LIN {X 0,Y 459.073,Z 809.06,A -85,B 0,C 180,E1 14501.398,E2 14501.398} C_VEL
LIN {X 0,Y 458.818,Z 809.06,A -85,B 0,C 180,E1 14507.25,E2 14507.25} C_VEL
LIN {X 0,Y 458.467,Z 809.06,A -85,B 0,C 180,E1 14513.306,E2 14513.306} C_VEL
LIN {X 0,Y 458.275,Z 809.06,A -85,B 0,C 180,E1 14519.651,E2 14519.651} C_VEL
LIN {X 0,Y 458.077,Z 809.06,A -85,B 0,C 180,E1 14526.434,E2 14526.434} C_VEL
LIN {X 0,Y 458.07,Z 809.06,A -85,B 0,C 180,E1 14531.291,E2 14531.291} C_VEL
LIN {X 0,Y 458.072,Z 809.06,A -85,B 0,C 180,E1 14536.54,E2 14536.54} C_VEL
LIN {X 0,Y 458,Z 809.06,A -85,B 0,C 180,E1 14542.368,E2 14542.368} C_VEL
LIN {X 0,Y 458.221,Z 809.06,A -85,B 0,C 180,E1 14549.039,E2 14549.039} C_VEL
LIN {X 0,Y 458.429,Z 809.06,A -85,B 0,C 180,E1 14554.63,E2 14554.63} C_VEL
LIN {X 0,Y 458.704,Z 809.06,A -85,B 0,C 180,E1 14560.768,E2 14560.768} C_VEL
LIN {X 0,Y 458.946,Z 809.06,A -85,B 0,C 180,E1 14566.677,E2 14566.677} C_VEL
LIN {X 0,Y 459.248,Z 809.06,A -85,B 0,C 180,E1 14573.134,E2 14573.134} C_VEL
LIN {X 0,Y 459.567,Z 809.06,A -85,B 0,C 180,E1 14578.117,E2 14578.117} C_VEL
LIN {X 0,Y 459.486,Z 809.06,A -85,B 0,C 180,E1 14583.772,E2 14583.772} C_VEL
LIN {X 0,Y 459.188,Z 809.06,A -85,B 0,C 180,E1 14589.471,E2 14589.471} C_VEL
LIN {X 0,Y 458.841,Z 809.06,A -85,B 0,C 180,E1 14595.275,E2 14595.275} C_VEL
LIN {X 0,Y 458.62,Z 809.313,A -85,B 0,C 180,E1 14601.041,E2 14601.041} C_VEL
LIN {X 0,Y 460.727,Z 814.529,A -85,B 0,C 180,E1 14601.677,E2 14601.677} C_VEL
LIN {X 0,Y 463.517,Z 818.136,A -85,B 0,C 180,E1 14602.358,E2 14602.358} C_VEL
LIN {X 0,Y 484.639,Z 848.609,A -85,B 0,C 180,E1 14607.191,E2 14607.191} C_VEL
LIN {X 0,Y 509.827,Z 888.021,A -85,B 0,C 180,E1 14612.178,E2 14612.178} C_VEL
LIN {X 0,Y 531.176,Z 928.04,A -85,B 0,C 180,E1 14616.332,E2 14616.332} C_VEL
LIN {X 0,Y 533.852,Z 935.082,A -85,B 0,C 180,E1 14616.915,E2 14616.915} C_VEL
LIN {X 0,Y 525.994,Z 983.884,A -85,B 0,C 180,E1 14618.511,E2 14618.511} C_VEL
LIN {X 0,Y 516.792,Z 1031.445,A -85,B 0,C 180,E1 14620.799,E2 14620.799} C_VEL
LIN {X 0,Y 506.374,Z 1076.578,A -85,B 0,C 180,E1 14623.742,E2 14623.742} C_VEL
LIN {X 0,Y 495.446,Z 1119.708,A -85,B 0,C 180,E1 14627.415,E2 14627.415} C_VEL
LIN {X 0,Y 484.874,Z 1160.046,A -85,B 0,C 180,E1 14631.936,E2 14631.936} C_VEL
LIN {X 0,Y 476.093,Z 1194.068,A -85,B 0,C 180,E1 14636.796,E2 14636.796} C_VEL
LIN {X 0,Y 468.636,Z 1225.613,A -85,B 0,C 180,E1 14642.62,E2 14642.62} C_VEL
LIN {X 0,Y 464.052,Z 1248.469,A -85,B 0,C 180,E1 14648.117,E2 14648.117} C_VEL
LIN {X 0,Y 461.344,Z 1266.286,A -85,B 0,C 180,E1 14653.827,E2 14653.827} C_VEL
LIN {X 0,Y 459.993,Z 1278.774,A -85,B 0,C 180,E1 14659.554,E2 14659.554} C_VEL
LIN {X 0,Y 459.672,Z 1284.621,A -85,B 0,C 180,E1 14664.333,E2 14664.333} C_VEL
LIN {X 0,Y 459.56,Z 1286.34,A -85,B 0,C 180,E1 14667.341,E2 14667.341} C_VEL
LIN {X 0,Y 457.078,Z 1286.869,A -85,B 0,C 180,E1 14668.953,E2 14668.953} C_VEL
LIN {X 0,Y 451.946,Z 1286.314,A -85,B 0,C 180,E1 14671.378,E2 14671.378} C_VEL
LIN {X 0,Y 451.892,Z 1286.241,A -85,B 0,C 180,E1 14671.658,E2 14671.658} C_VEL
LIN {X 0,Y 451.956,Z 1281.773,A -85,B 0,C 180,E1 14677.677,E2 14677.677} C_VEL
LIN {X 0,Y 452.703,Z 1272.747,A -85,B 0,C 180,E1 14683.013,E2 14683.013} C_VEL
LIN {X 0,Y 454.412,Z 1258.506,A -85,B 0,C 180,E1 14688.449,E2 14688.449} C_VEL
LIN {X 0,Y 457.628,Z 1239.088,A -85,B 0,C 180,E1 14693.825,E2 14693.825} C_VEL
LIN {X 0,Y 462.745,Z 1212.947,A -85,B 0,C 180,E1 14699.319,E2 14699.319} C_VEL
LIN {X 0,Y 469.367,Z 1182.336,A -85,B 0,C 180,E1 14704.276,E2 14704.276} C_VEL
LIN {X 0,Y 477.757,Z 1144.374,A -85,B 0,C 180,E1 14709.083,E2 14709.083} C_VEL
LIN {X 0,Y 486.62,Z 1104.059,A -85,B 0,C 180,E1 14713.08,E2 14713.08} C_VEL
LIN {X 0,Y 496.53,Z 1056.093,A -85,B 0,C 180,E1 14716.748,E2 14716.748} C_VEL
LIN {X 0,Y 505.91,Z 1006.434,A -85,B 0,C 180,E1 14719.639,E2 14719.639} C_VEL
LIN {X 0,Y 515.783,Z 948.619,A -85,B 0,C 180,E1 14722.104,E2 14722.104} C_VEL
LIN {X 0,Y 517.829,Z 935.284,A -85,B 0,C 180,E1 14722.543,E2 14722.543} C_VEL
LIN {X 0,Y 507.618,Z 899.519,A -85,B 0,C 180,E1 14726.042,E2 14726.042} C_VEL
LIN {X 0,Y 505.964,Z 885.962,A -85,B 0,C 180,E1 14728.048,E2 14728.048} C_VEL
LIN {X 0,Y 505.994,Z 884.666,A -85,B 0,C 180,E1 14728.412,E2 14728.412} C_VEL
LIN {X 0,Y 504.35,Z 894.37,A -85,B 0,C 180,E1 14730.603,E2 14730.603} C_VEL
LIN {X 0,Y 507.893,Z 921.665,A -85,B 0,C 180,E1 14734.702,E2 14734.702} C_VEL
LIN {X 0,Y 511.089,Z 938.057,A -85,B 0,C 180,E1 14736.979,E2 14736.979} C_VEL
LIN {X 0,Y 500.885,Z 977.012,A -85,B 0,C 180,E1 14740.046,E2 14740.046} C_VEL
LIN {X 0,Y 489.61,Z 1013.591,A -85,B 0,C 180,E1 14743.873,E2 14743.873} C_VEL
LIN {X 0,Y 479.089,Z 1044.899,A -85,B 0,C 180,E1 14748.178,E2 14748.178} C_VEL
LIN {X 0,Y 468.845,Z 1074.319,A -85,B 0,C 180,E1 14753.523,E2 14753.523} C_VEL
LIN {X 0,Y 460.77,Z 1098.348,A -85,B 0,C 180,E1 14759.515,E2 14759.515} C_VEL
LIN {X 0,Y 455.737,Z 1115.395,A -85,B 0,C 180,E1 14765.369,E2 14765.369} C_VEL
LIN {X 0,Y 453.06,Z 1127.764,A -85,B 0,C 180,E1 14771.542,E2 14771.542} C_VEL
LIN {X 0,Y 451.778,Z 1135.121,A -85,B 0,C 180,E1 14777.517,E2 14777.517} C_VEL
LIN {X 0,Y 450.908,Z 1138.251,A -85,B 0,C 180,E1 14783.71,E2 14783.71} C_VEL
LIN {X 0,Y 451.301,Z 1136.637,A -85,B 0,C 180,E1 14790.146,E2 14790.146} C_VEL
LIN {X 0,Y 452.358,Z 1131.437,A -85,B 0,C 180,E1 14795.485,E2 14795.485} C_VEL
LIN {X 0,Y 453.774,Z 1122.657,A -85,B 0,C 180,E1 14800.796,E2 14800.796} C_VEL
LIN {X 0,Y 456.953,Z 1108.165,A -85,B 0,C 180,E1 14806.673,E2 14806.673} C_VEL
LIN {X 0,Y 462.638,Z 1088.104,A -85,B 0,C 180,E1 14812.52,E2 14812.52} C_VEL
LIN {X 0,Y 470.74,Z 1062.034,A -85,B 0,C 180,E1 14818.105,E2 14818.105} C_VEL
LIN {X 0,Y 480.037,Z 1033.327,A -85,B 0,C 180,E1 14822.802,E2 14822.802} C_VEL
LIN {X 0,Y 491.09,Z 998.255,A -85,B 0,C 180,E1 14827.17,E2 14827.17} C_VEL
LIN {X 0,Y 502.007,Z 960.535,A -85,B 0,C 180,E1 14830.786,E2 14830.786} C_VEL
LIN {X 0,Y 508.357,Z 935.557,A -85,B 0,C 180,E1 14832.715,E2 14832.715} C_VEL
LIN {X 0,Y 498.985,Z 904.371,A -85,B 0,C 180,E1 14836.88,E2 14836.88} C_VEL
LIN {X 0,Y 485.509,Z 871.059,A -85,B 0,C 180,E1 14841.568,E2 14841.568} C_VEL
LIN {X 0,Y 469.62,Z 840.002,A -85,B 0,C 180,E1 14846.422,E2 14846.422} C_VEL
LIN {X 0,Y 454.416,Z 815.01,A -85,B 0,C 180,E1 14850.902,E2 14850.902} C_VEL
LIN {X 0,Y 451.695,Z 809.882,A -85,B 0,C 180,E1 14851.745,E2 14851.745} C_VEL
LIN {X 0,Y 451.507,Z 809.06,A -85,B 0,C 180,E1 14853.846,E2 14853.846} C_VEL
LIN {X 0,Y 451.253,Z 809.06,A -85,B 0,C 180,E1 14859.646,E2 14859.646} C_VEL
LIN {X 0,Y 450.953,Z 809.06,A -85,B 0,C 180,E1 14865.557,E2 14865.557} C_VEL
LIN {X 0,Y 450.624,Z 809.06,A -85,B 0,C 180,E1 14871.653,E2 14871.653} C_VEL
LIN {X 0,Y 450.391,Z 809.06,A -85,B 0,C 180,E1 14878.023,E2 14878.023} C_VEL
LIN {X 0,Y 450.197,Z 809.06,A -85,B 0,C 180,E1 14884.801,E2 14884.801} C_VEL
LIN {X 0,Y 450.133,Z 809.06,A -85,B 0,C 180,E1 14889.639,E2 14889.639} C_VEL
LIN {X 0,Y 450.084,Z 809.06,A -85,B 0,C 180,E1 14895.172,E2 14895.172} C_VEL
LIN {X 0,Y 450.079,Z 809.06,A -85,B 0,C 180,E1 14900.562,E2 14900.562} C_VEL
LIN {X 0,Y 450.156,Z 809.06,A -85,B 0,C 180,E1 14907.068,E2 14907.068} C_VEL
LIN {X 0,Y 450.393,Z 809.06,A -85,B 0,C 180,E1 14911.988,E2 14911.988} C_VEL
LIN {X 0,Y 450.672,Z 809.06,A -85,B 0,C 180,E1 14918.359,E2 14918.359} C_VEL
LIN {X 0,Y 450.885,Z 809.06,A -85,B 0,C 180,E1 14924.45,E2 14924.45} C_VEL
LIN {X 0,Y 451.262,Z 809.06,A -85,B 0,C 180,E1 14930.363,E2 14930.363} C_VEL
LIN {X 0,Y 451.566,Z 809.06,A -85,B 0,C 180,E1 14936.164,E2 14936.164} C_VEL
LIN {X 0,Y 451.767,Z 809.06,A -85,B 0,C 180,E1 14941.917,E2 14941.917} C_VEL
LIN {X 0,Y 451.343,Z 809.06,A -85,B 0,C 180,E1 14947.696,E2 14947.696} C_VEL
LIN {X 0,Y 451.023,Z 809.06,A -85,B 0,C 180,E1 14953.661,E2 14953.661} C_VEL
LIN {X 0,Y 450.817,Z 809.82,A -85,B 0,C 180,E1 14959.392,E2 14959.392} C_VEL
LIN {X 0,Y 453.497,Z 815.064,A -85,B 0,C 180,E1 14960.162,E2 14960.162} C_VEL
LIN {X 0,Y 455.851,Z 818.218,A -85,B 0,C 180,E1 14960.792,E2 14960.792} C_VEL
LIN {X 0,Y 474.523,Z 845.268,A -85,B 0,C 180,E1 14965.35,E2 14965.35} C_VEL
LIN {X 0,Y 499.268,Z 883.021,A -85,B 0,C 180,E1 14970.523,E2 14970.523} C_VEL
LIN {X 0,Y 521.728,Z 923.677,A -85,B 0,C 180,E1 14975.016,E2 14975.016} C_VEL
LIN {X 0,Y 528.094,Z 937.427,A -85,B 0,C 180,E1 14976.349,E2 14976.349} C_VEL
LIN {X 0,Y 519.566,Z 988.021,A -85,B 0,C 180,E1 14978.079,E2 14978.079} C_VEL
LIN {X 0,Y 510.247,Z 1034.148,A -85,B 0,C 180,E1 14980.364,E2 14980.364} C_VEL
LIN {X 0,Y 498.846,Z 1081.49,A -85,B 0,C 180,E1 14983.565,E2 14983.565} C_VEL
LIN {X 0,Y 487.789,Z 1123.072,A -85,B 0,C 180,E1 14987.26,E2 14987.26} C_VEL
LIN {X 0,Y 477.179,Z 1162.261,A -85,B 0,C 180,E1 14991.785,E2 14991.785} C_VEL
LIN {X 0,Y 468.218,Z 1195.558,A -85,B 0,C 180,E1 14996.718,E2 14996.718} C_VEL
LIN {X 0,Y 461.085,Z 1224.685,A -85,B 0,C 180,E1 15002.228,E2 15002.228} C_VEL
LIN {X 0,Y 456.204,Z 1248.219,A -85,B 0,C 180,E1 15008.033,E2 15008.033} C_VEL
LIN {X 0,Y 453.562,Z 1265.022,A -85,B 0,C 180,E1 15013.542,E2 15013.542} C_VEL
LIN {X 0,Y 452.345,Z 1275.819,A -85,B 0,C 180,E1 15018.43,E2 15018.43} C_VEL
LIN {X 0,Y 451.967,Z 1281.836,A -85,B 0,C 180,E1 15022.307,E2 15022.307} C_VEL
LIN {X 0,Y 451.745,Z 1286.16,A -85,B 0,C 180,E1 15028.075,E2 15028.075} C_VEL
LIN {X 0,Y 451.892,Z 1286.241,A -85,B 0,C 180,E1 15031.658,E2 15031.658} C_VEL
LIN {X 0,Y 449.493,Z 1285.263,A -85,B 0,C 180,E1 15033.286,E2 15033.286} C_VEL
LIN {X 0,Y 444.015,Z 1282.245,A -85,B 0,C 180,E1 15036.001,E2 15036.001} C_VEL
LIN {X 0,Y 444.472,Z 1275.955,A -85,B 0,C 180,E1 15040.768,E2 15040.768} C_VEL
LIN {X 0,Y 445.669,Z 1264.065,A -85,B 0,C 180,E1 15046.235,E2 15046.235} C_VEL
LIN {X 0,Y 448.266,Z 1246.87,A -85,B 0,C 180,E1 15051.756,E2 15051.756} C_VEL
LIN {X 0,Y 452.324,Z 1224.795,A -85,B 0,C 180,E1 15057.066,E2 15057.066} C_VEL
LIN {X 0,Y 458.574,Z 1196.263,A -85,B 0,C 180,E1 15062.373,E2 15062.373} C_VEL
LIN {X 0,Y 466.395,Z 1162.049,A -85,B 0,C 180,E1 15067.294,E2 15067.294} C_VEL
LIN {X 0,Y 475.604,Z 1121.839,A -85,B 0,C 180,E1 15071.841,E2 15071.841} C_VEL
LIN {X 0,Y 485.521,Z 1077.379,A -85,B 0,C 180,E1 15075.699,E2 15075.699} C_VEL
LIN {X 0,Y 495.288,Z 1029.918,A -85,B 0,C 180,E1 15078.903,E2 15078.903} C_VEL
LIN {X 0,Y 504.786,Z 979.028,A -85,B 0,C 180,E1 15081.496,E2 15081.496} C_VEL
LIN {X 0,Y 511.598,Z 937.834,A -85,B 0,C 180,E1 15083.138,E2 15083.138} C_VEL
LIN {X 0,Y 503.854,Z 906.093,A -85,B 0,C 180,E1 15086.378,E2 15086.378} C_VEL
LIN {X 0,Y 503.15,Z 893.729,A -85,B 0,C 180,E1 15088.205,E2 15088.205} C_VEL
LIN {X 0,Y 503.056,Z 893.125,A -85,B 0,C 180,E1 15088.555,E2 15088.555} C_VEL
LIN {X 0,Y 500.921,Z 904.138,A -85,B 0,C 180,E1 15090.847,E2 15090.847} C_VEL
LIN {X 0,Y 505.503,Z 941.412,A -85,B 0,C 180,E1 15096.443,E2 15096.443} C_VEL
LIN {X 0,Y 494.875,Z 980.106,A -85,B 0,C 180,E1 15099.56,E2 15099.56} C_VEL
LIN {X 0,Y 483.27,Z 1016.326,A -85,B 0,C 180,E1 15103.422,E2 15103.422} C_VEL
LIN {X 0,Y 472.262,Z 1047.658,A -85,B 0,C 180,E1 15107.819,E2 15107.819} C_VEL
LIN {X 0,Y 462.173,Z 1075.434,A -85,B 0,C 180,E1 15112.957,E2 15112.957} C_VEL
LIN {X 0,Y 454.375,Z 1097.488,A -85,B 0,C 180,E1 15118.443,E2 15118.443} C_VEL
LIN {X 0,Y 448.592,Z 1115.922,A -85,B 0,C 180,E1 15124.658,E2 15124.658} C_VEL
LIN {X 0,Y 445.664,Z 1127.858,A -85,B 0,C 180,E1 15130.543,E2 15130.543} C_VEL
LIN {X 0,Y 444.326,Z 1134.908,A -85,B 0,C 180,E1 15135.786,E2 15135.786} C_VEL
LIN {X 0,Y 443.237,Z 1139.205,A -85,B 0,C 180,E1 15142.023,E2 15142.023} C_VEL
LIN {X 0,Y 443.275,Z 1138.821,A -85,B 0,C 180,E1 15148.503,E2 15148.503} C_VEL
LIN {X 0,Y 444.258,Z 1134.571,A -85,B 0,C 180,E1 15153.963,E2 15153.963} C_VEL
LIN {X 0,Y 445.795,Z 1125.624,A -85,B 0,C 180,E1 15160.089,E2 15160.089} C_VEL
LIN {X 0,Y 448.665,Z 1112.355,A -85,B 0,C 180,E1 15165.931,E2 15165.931} C_VEL
LIN {X 0,Y 454.479,Z 1092.107,A -85,B 0,C 180,E1 15172.18,E2 15172.18} C_VEL
LIN {X 0,Y 461.863,Z 1069.016,A -85,B 0,C 180,E1 15177.464,E2 15177.464} C_VEL
LIN {X 0,Y 472.192,Z 1038.17,A -85,B 0,C 180,E1 15182.773,E2 15182.773} C_VEL
LIN {X 0,Y 482.736,Z 1006.027,A -85,B 0,C 180,E1 15186.992,E2 15186.992} C_VEL
LIN {X 0,Y 494.625,Z 966.727,A -85,B 0,C 180,E1 15190.932,E2 15190.932} C_VEL
LIN {X 0,Y 502.079,Z 938.758,A -85,B 0,C 180,E1 15193.169,E2 15193.169} C_VEL
LIN {X 0,Y 492.985,Z 907.827,A -85,B 0,C 180,E1 15197.393,E2 15197.393} C_VEL
LIN {X 0,Y 480.041,Z 875.321,A -85,B 0,C 180,E1 15202.092,E2 15202.092} C_VEL
LIN {X 0,Y 464.938,Z 845.25,A -85,B 0,C 180,E1 15206.922,E2 15206.922} C_VEL
LIN {X 0,Y 450.629,Z 821.483,A -85,B 0,C 180,E1 15211.276,E2 15211.276} C_VEL
LIN {X 0,Y 446.35,Z 814.995,A -85,B 0,C 180,E1 15212.615,E2 15212.615} C_VEL
LIN {X 0,Y 443.672,Z 810.022,A -85,B 0,C 180,E1 15213.486,E2 15213.486} C_VEL
LIN {X 0,Y 443.596,Z 809.06,A -85,B 0,C 180,E1 15213.914,E2 15213.914} C_VEL
LIN {X 0,Y 443.332,Z 809.06,A -85,B 0,C 180,E1 15219.82,E2 15219.82} C_VEL
LIN {X 0,Y 443.006,Z 809.06,A -85,B 0,C 180,E1 15225.843,E2 15225.843} C_VEL
LIN {X 0,Y 442.652,Z 809.06,A -85,B 0,C 180,E1 15232.064,E2 15232.064} C_VEL
LIN {X 0,Y 442.457,Z 809.06,A -85,B 0,C 180,E1 15238.572,E2 15238.572} C_VEL
LIN {X 0,Y 442.267,Z 809.06,A -85,B 0,C 180,E1 15245.518,E2 15245.518} C_VEL
LIN {X 0,Y 442.109,Z 809.06,A -85,B 0,C 180,E1 15251.247,E2 15251.247} C_VEL
LIN {X 0,Y 442.089,Z 809.06,A -85,B 0,C 180,E1 15256.878,E2 15256.878} C_VEL
LIN {X 0,Y 442.109,Z 809.06,A -85,B 0,C 180,E1 15262.036,E2 15262.036} C_VEL
LIN {X 0,Y 442.287,Z 809.06,A -85,B 0,C 180,E1 15268.677,E2 15268.677} C_VEL
LIN {X 0,Y 442.506,Z 809.06,A -85,B 0,C 180,E1 15273.648,E2 15273.648} C_VEL
LIN {X 0,Y 442.832,Z 809.06,A -85,B 0,C 180,E1 15280.05,E2 15280.05} C_VEL
LIN {X 0,Y 443.096,Z 809.06,A -85,B 0,C 180,E1 15286.191,E2 15286.191} C_VEL
LIN {X 0,Y 443.431,Z 809.06,A -85,B 0,C 180,E1 15292.167,E2 15292.167} C_VEL
LIN {X 0,Y 443.778,Z 809.06,A -85,B 0,C 180,E1 15298.05,E2 15298.05} C_VEL
LIN {X 0,Y 443.661,Z 809.06,A -85,B 0,C 180,E1 15303.906,E2 15303.906} C_VEL
LIN {X 0,Y 443.324,Z 809.06,A -85,B 0,C 180,E1 15309.813,E2 15309.813} C_VEL
LIN {X 0,Y 442.959,Z 809.06,A -85,B 0,C 180,E1 15315.837,E2 15315.837} C_VEL
LIN {X 0,Y 442.983,Z 809.793,A -85,B 0,C 180,E1 15317.595,E2 15317.595} C_VEL
LIN {X 0,Y 445.55,Z 814.971,A -85,B 0,C 180,E1 15318.432,E2 15318.432} C_VEL
LIN {X 0,Y 447.849,Z 817.771,A -85,B 0,C 180,E1 15319.064,E2 15319.064} C_VEL
LIN {X 0,Y 470.21,Z 850.079,A -85,B 0,C 180,E1 15324.734,E2 15324.734} C_VEL
LIN {X 0,Y 495.465,Z 889.163,A -85,B 0,C 180,E1 15330.149,E2 15330.149} C_VEL
LIN {X 0,Y 516.651,Z 928.45,A -85,B 0,C 180,E1 15334.588,E2 15334.588} C_VEL
LIN {X 0,Y 522.067,Z 941.841,A -85,B 0,C 180,E1 15335.852,E2 15335.852} C_VEL
LIN {X 0,Y 513.617,Z 989.596,A -85,B 0,C 180,E1 15337.526,E2 15337.526} C_VEL
LIN {X 0,Y 504.319,Z 1033.697,A -85,B 0,C 180,E1 15339.742,E2 15339.742} C_VEL
LIN {X 0,Y 492.597,Z 1081.043,A -85,B 0,C 180,E1 15342.963,E2 15342.963} C_VEL
LIN {X 0,Y 481.077,Z 1122.731,A -85,B 0,C 180,E1 15346.714,E2 15346.714} C_VEL
LIN {X 0,Y 470.325,Z 1161.163,A -85,B 0,C 180,E1 15351.199,E2 15351.199} C_VEL
LIN {X 0,Y 461.155,Z 1194.105,A -85,B 0,C 180,E1 15356.14,E2 15356.14} C_VEL
LIN {X 0,Y 453.425,Z 1224.352,A -85,B 0,C 180,E1 15361.949,E2 15361.949} C_VEL
LIN {X 0,Y 448.54,Z 1246.928,A -85,B 0,C 180,E1 15367.637,E2 15367.637} C_VEL
LIN {X 0,Y 445.798,Z 1263.758,A -85,B 0,C 180,E1 15373.247,E2 15373.247} C_VEL
LIN {X 0,Y 444.533,Z 1274.57,A -85,B 0,C 180,E1 15378.224,E2 15378.224} C_VEL
LIN {X 0,Y 444.149,Z 1280.597,A -85,B 0,C 180,E1 15382.171,E2 15382.171} C_VEL
LIN {X 0,Y 443.957,Z 1284.881,A -85,B 0,C 180,E1 15388.042,E2 15388.042} C_VEL
LIN {X 0,Y 444.14,Z 1284.887,A -85,B 0,C 180,E1 15391.942,E2 15391.942} C_VEL
LIN {X 0,Y 444.015,Z 1282.245,A -85,B 0,C 180,E1 15396.001,E2 15396.001} C_VEL
LIN {X 0,Y 440.201,Z 1279.247,A -85,B 0,C 180,E1 15398.182,E2 15398.182} C_VEL
LIN {X 0,Y 436.562,Z 1275.412,A -85,B 0,C 180,E1 15400.386,E2 15400.386} C_VEL
LIN {X 0,Y 437.772,Z 1263.857,A -85,B 0,C 180,E1 15406.021,E2 15406.021} C_VEL
LIN {X 0,Y 440.298,Z 1246.946,A -85,B 0,C 180,E1 15411.641,E2 15411.641} C_VEL
LIN {X 0,Y 444.504,Z 1224.438,A -85,B 0,C 180,E1 15417.204,E2 15417.204} C_VEL
LIN {X 0,Y 450.946,Z 1195.849,A -85,B 0,C 180,E1 15422.645,E2 15422.645} C_VEL
LIN {X 0,Y 458.759,Z 1162.661,A -85,B 0,C 180,E1 15427.537,E2 15427.537} C_VEL
LIN {X 0,Y 468.449,Z 1121.839,A -85,B 0,C 180,E1 15432.249,E2 15432.249} C_VEL
LIN {X 0,Y 478.271,Z 1079.418,A -85,B 0,C 180,E1 15436.037,E2 15436.037} C_VEL
LIN {X 0,Y 488.887,Z 1029.944,A -85,B 0,C 180,E1 15439.453,E2 15439.453} C_VEL
LIN {X 0,Y 498.797,Z 980.089,A -85,B 0,C 180,E1 15442.067,E2 15442.067} C_VEL
LIN {X 0,Y 505.765,Z 940.787,A -85,B 0,C 180,E1 15443.72,E2 15443.72} C_VEL
LIN {X 0,Y 500.141,Z 914.05,A -85,B 0,C 180,E1 15446.539,E2 15446.539} C_VEL
LIN {X 0,Y 500.095,Z 901.629,A -85,B 0,C 180,E1 15448.347,E2 15448.347} C_VEL
LIN {X 0,Y 498.114,Z 906.584,A -85,B 0,C 180,E1 15449.714,E2 15449.714} C_VEL
LIN {X 0,Y 497.592,Z 925.176,A -85,B 0,C 180,E1 15452.903,E2 15452.903} C_VEL
LIN {X 0,Y 500.008,Z 945.197,A -85,B 0,C 180,E1 15455.922,E2 15455.922} C_VEL
LIN {X 0,Y 488.917,Z 983.362,A -85,B 0,C 180,E1 15459.063,E2 15459.063} C_VEL
LIN {X 0,Y 476.416,Z 1020.906,A -85,B 0,C 180,E1 15463.177,E2 15463.177} C_VEL
LIN {X 0,Y 464.656,Z 1052.627,A -85,B 0,C 180,E1 15467.82,E2 15467.82} C_VEL
LIN {X 0,Y 454.737,Z 1078.75,A -85,B 0,C 180,E1 15472.841,E2 15472.841} C_VEL
LIN {X 0,Y 446.004,Z 1102.601,A -85,B 0,C 180,E1 15479.077,E2 15479.077} C_VEL
LIN {X 0,Y 440.81,Z 1118.375,A -85,B 0,C 180,E1 15484.766,E2 15484.766} C_VEL
LIN {X 0,Y 437.872,Z 1129.945,A -85,B 0,C 180,E1 15490.733,E2 15490.733} C_VEL
LIN {X 0,Y 436.506,Z 1136.694,A -85,B 0,C 180,E1 15496.076,E2 15496.076} C_VEL
LIN {X 0,Y 435.394,Z 1140.688,A -85,B 0,C 180,E1 15502.441,E2 15502.441} C_VEL
LIN {X 0,Y 435.305,Z 1140.637,A -85,B 0,C 180,E1 15506.823,E2 15506.823} C_VEL
LIN {X 0,Y 436.122,Z 1137.572,A -85,B 0,C 180,E1 15512.293,E2 15512.293} C_VEL
LIN {X 0,Y 437.542,Z 1130.055,A -85,B 0,C 180,E1 15518.432,E2 15518.432} C_VEL
LIN {X 0,Y 440.183,Z 1117.221,A -85,B 0,C 180,E1 15524.779,E2 15524.779} C_VEL
LIN {X 0,Y 445.254,Z 1099.657,A -85,B 0,C 180,E1 15530.831,E2 15530.831} C_VEL
LIN {X 0,Y 452.657,Z 1076.645,A -85,B 0,C 180,E1 15536.564,E2 15536.564} C_VEL
LIN {X 0,Y 462.482,Z 1048.373,A -85,B 0,C 180,E1 15541.898,E2 15541.898} C_VEL
LIN {X 0,Y 473.813,Z 1014.875,A -85,B 0,C 180,E1 15546.631,E2 15546.631} C_VEL
LIN {X 0,Y 485.462,Z 978.695,A -85,B 0,C 180,E1 15550.558,E2 15550.558} C_VEL
LIN {X 0,Y 495.615,Z 941.523,A -85,B 0,C 180,E1 15553.692,E2 15553.692} C_VEL
LIN {X 0,Y 486.974,Z 911.319,A -85,B 0,C 180,E1 15557.917,E2 15557.917} C_VEL
LIN {X 0,Y 474.462,Z 879.124,A -85,B 0,C 180,E1 15562.689,E2 15562.689} C_VEL
LIN {X 0,Y 458.779,Z 847.512,A -85,B 0,C 180,E1 15567.902,E2 15567.902} C_VEL
LIN {X 0,Y 445.788,Z 826.374,A -85,B 0,C 180,E1 15571.988,E2 15571.988} C_VEL
LIN {X 0,Y 438.569,Z 815.198,A -85,B 0,C 180,E1 15574.339,E2 15574.339} C_VEL
LIN {X 0,Y 435.742,Z 810.392,A -85,B 0,C 180,E1 15575.293,E2 15575.293} C_VEL
LIN {X 0,Y 435.621,Z 809.06,A -85,B 0,C 180,E1 15575.432,E2 15575.432} C_VEL
LIN {X 0,Y 435.272,Z 809.06,A -85,B 0,C 180,E1 15582.03,E2 15582.03} C_VEL
LIN {X 0,Y 434.961,Z 809.06,A -85,B 0,C 180,E1 15588.228,E2 15588.228} C_VEL
LIN {X 0,Y 434.573,Z 809.06,A -85,B 0,C 180,E1 15595.312,E2 15595.312} C_VEL
LIN {X 0,Y 434.412,Z 809.06,A -85,B 0,C 180,E1 15601.46,E2 15601.46} C_VEL
LIN {X 0,Y 434.221,Z 809.06,A -85,B 0,C 180,E1 15606.838,E2 15606.838} C_VEL
LIN {X 0,Y 434.198,Z 809.06,A -85,B 0,C 180,E1 15613.048,E2 15613.048} C_VEL
LIN {X 0,Y 434.164,Z 809.06,A -85,B 0,C 180,E1 15618.606,E2 15618.606} C_VEL
LIN {X 0,Y 434.196,Z 809.06,A -85,B 0,C 180,E1 15623.731,E2 15623.731} C_VEL
LIN {X 0,Y 434.42,Z 809.06,A -85,B 0,C 180,E1 15630.426,E2 15630.426} C_VEL
LIN {X 0,Y 434.632,Z 809.06,A -85,B 0,C 180,E1 15635.344,E2 15635.344} C_VEL
LIN {X 0,Y 434.96,Z 809.06,A -85,B 0,C 180,E1 15641.782,E2 15641.782} C_VEL
LIN {X 0,Y 435.254,Z 809.06,A -85,B 0,C 180,E1 15647.979,E2 15647.979} C_VEL
LIN {X 0,Y 435.625,Z 809.06,A -85,B 0,C 180,E1 15654.028,E2 15654.028} C_VEL
LIN {X 0,Y 436.103,Z 809.06,A -85,B 0,C 180,E1 15660.001,E2 15660.001} C_VEL
LIN {X 0,Y 435.647,Z 809.06,A -85,B 0,C 180,E1 15665.973,E2 15665.973} C_VEL
LIN {X 0,Y 435.264,Z 809.06,A -85,B 0,C 180,E1 15672.023,E2 15672.023} C_VEL
LIN {X 0,Y 435.058,Z 809.061,A -85,B 0,C 180,E1 15675.68,E2 15675.68} C_VEL
LIN {X 0,Y 437.031,Z 814.305,A -85,B 0,C 180,E1 15676.396,E2 15676.396} C_VEL
LIN {X 0,Y 440.172,Z 817.923,A -85,B 0,C 180,E1 15677.288,E2 15677.288} C_VEL
LIN {X 0,Y 459.035,Z 845.049,A -85,B 0,C 180,E1 15682.442,E2 15682.442} C_VEL
LIN {X 0,Y 481.736,Z 879.279,A -85,B 0,C 180,E1 15687.685,E2 15687.685} C_VEL
LIN {X 0,Y 502.019,Z 914.261,A -85,B 0,C 180,E1 15692.055,E2 15692.055} C_VEL
LIN {X 0,Y 516.35,Z 944.429,A -85,B 0,C 180,E1 15695.287,E2 15695.287} C_VEL
LIN {X 0,Y 507.645,Z 991.542,A -85,B 0,C 180,E1 15696.976,E2 15696.976} C_VEL
LIN {X 0,Y 497.505,Z 1037.282,A -85,B 0,C 180,E1 15699.357,E2 15699.357} C_VEL
LIN {X 0,Y 485.938,Z 1082.369,A -85,B 0,C 180,E1 15702.493,E2 15702.493} C_VEL
LIN {X 0,Y 474.142,Z 1123.455,A -85,B 0,C 180,E1 15706.269,E2 15706.269} C_VEL
LIN {X 0,Y 463.135,Z 1161.426,A -85,B 0,C 180,E1 15710.782,E2 15710.782} C_VEL
LIN {X 0,Y 453.642,Z 1194.337,A -85,B 0,C 180,E1 15715.836,E2 15715.836} C_VEL
LIN {X 0,Y 445.795,Z 1224.005,A -85,B 0,C 180,E1 15721.662,E2 15721.662} C_VEL
LIN {X 0,Y 440.502,Z 1247.679,A -85,B 0,C 180,E1 15727.843,E2 15727.843} C_VEL
LIN {X 0,Y 437.835,Z 1263.783,A -85,B 0,C 180,E1 15733.449,E2 15733.449} C_VEL
LIN {X 0,Y 436.52,Z 1275.089,A -85,B 0,C 180,E1 15739.016,E2 15739.016} C_VEL
LIN {X 0,Y 436.192,Z 1281.308,A -85,B 0,C 180,E1 15744.027,E2 15744.027} C_VEL
LIN {X 0,Y 436.288,Z 1284.002,A -85,B 0,C 180,E1 15749.992,E2 15749.992} C_VEL
LIN {X 0,Y 436.205,Z 1282.566,A -85,B 0,C 180,E1 15753.965,E2 15753.965} C_VEL
LIN {X 0,Y 436.421,Z 1277.971,A -85,B 0,C 180,E1 15758.657,E2 15758.657} C_VEL
LIN {X 0,Y 436.562,Z 1275.412,A -85,B 0,C 180,E1 15760.386,E2 15760.386} C_VEL
LIN {X 0,Y 435.505,Z 1273.375,A -85,B 0,C 180,E1 15761.497,E2 15761.497} C_VEL
LIN {X 0,Y 429.675,Z 1266.507,A -85,B 0,C 180,E1 15764.491,E2 15764.491} C_VEL
LIN {X 0,Y 429.66,Z 1265.852,A -85,B 0,C 180,E1 15764.773,E2 15764.773} C_VEL
LIN {X 0,Y 431.814,Z 1250.39,A -85,B 0,C 180,E1 15770.474,E2 15770.474} C_VEL
LIN {X 0,Y 435.614,Z 1229.748,A -85,B 0,C 180,E1 15776.07,E2 15776.07} C_VEL
LIN {X 0,Y 441.674,Z 1202.342,A -85,B 0,C 180,E1 15781.697,E2 15781.697} C_VEL
LIN {X 0,Y 449.75,Z 1168.938,A -85,B 0,C 180,E1 15787.008,E2 15787.008} C_VEL
LIN {X 0,Y 458.926,Z 1131.859,A -85,B 0,C 180,E1 15791.615,E2 15791.615} C_VEL
LIN {X 0,Y 469.237,Z 1088.849,A -85,B 0,C 180,E1 15795.764,E2 15795.764} C_VEL
LIN {X 0,Y 480.185,Z 1041.084,A -85,B 0,C 180,E1 15799.339,E2 15799.339} C_VEL
LIN {X 0,Y 491.732,Z 986.539,A -85,B 0,C 180,E1 15802.408,E2 15802.408} C_VEL
LIN {X 0,Y 500.19,Z 944.354,A -85,B 0,C 180,E1 15804.242,E2 15804.242} C_VEL
LIN {X 0,Y 496.217,Z 918.391,A -85,B 0,C 180,E1 15807.169,E2 15807.169} C_VEL
LIN {X 0,Y 496.758,Z 910.263,A -85,B 0,C 180,E1 15808.384,E2 15808.384} C_VEL
LIN {X 0,Y 495.332,Z 912.721,A -85,B 0,C 180,E1 15809.243,E2 15809.243} C_VEL
LIN {X 0,Y 493.21,Z 930.066,A -85,B 0,C 180,E1 15812.384,E2 15812.384} C_VEL
LIN {X 0,Y 494.592,Z 949.106,A -85,B 0,C 180,E1 15815.379,E2 15815.379} C_VEL
LIN {X 0,Y 482.697,Z 987.752,A -85,B 0,C 180,E1 15818.66,E2 15818.66} C_VEL
LIN {X 0,Y 470.165,Z 1023.776,A -85,B 0,C 180,E1 15822.706,E2 15822.706} C_VEL
LIN {X 0,Y 457.508,Z 1056.505,A -85,B 0,C 180,E1 15827.627,E2 15827.627} C_VEL
LIN {X 0,Y 446.865,Z 1083.007,A -85,B 0,C 180,E1 15832.959,E2 15832.959} C_VEL
LIN {X 0,Y 438.879,Z 1104.034,A -85,B 0,C 180,E1 15838.628,E2 15838.628} C_VEL
LIN {X 0,Y 433.217,Z 1120.349,A -85,B 0,C 180,E1 15844.664,E2 15844.664} C_VEL
LIN {X 0,Y 429.995,Z 1132.471,A -85,B 0,C 180,E1 15851.204,E2 15851.204} C_VEL
LIN {X 0,Y 428.668,Z 1138.497,A -85,B 0,C 180,E1 15856.378,E2 15856.378} C_VEL
LIN {X 0,Y 427.539,Z 1142.021,A -85,B 0,C 180,E1 15862.876,E2 15862.876} C_VEL
LIN {X 0,Y 427.548,Z 1141.602,A -85,B 0,C 180,E1 15867.944,E2 15867.944} C_VEL
LIN {X 0,Y 428.749,Z 1136.882,A -85,B 0,C 180,E1 15874.323,E2 15874.323} C_VEL
LIN {X 0,Y 430.373,Z 1128.239,A -85,B 0,C 180,E1 15880.402,E2 15880.402} C_VEL
LIN {X 0,Y 433.469,Z 1115.443,A -85,B 0,C 180,E1 15886.312,E2 15886.312} C_VEL
LIN {X 0,Y 439.559,Z 1095.698,A -85,B 0,C 180,E1 15892.643,E2 15892.643} C_VEL
LIN {X 0,Y 447.827,Z 1071.814,A -85,B 0,C 180,E1 15898.328,E2 15898.328} C_VEL
LIN {X 0,Y 458.36,Z 1042.127,A -85,B 0,C 180,E1 15903.58,E2 15903.58} C_VEL
LIN {X 0,Y 470.081,Z 1008.806,A -85,B 0,C 180,E1 15908.082,E2 15908.082} C_VEL
LIN {X 0,Y 482.392,Z 970.197,A -85,B 0,C 180,E1 15912.025,E2 15912.025} C_VEL
LIN {X 0,Y 489.324,Z 944.613,A -85,B 0,C 180,E1 15914.178,E2 15914.178} C_VEL
LIN {X 0,Y 480.993,Z 914.831,A -85,B 0,C 180,E1 15918.455,E2 15918.455} C_VEL
LIN {X 0,Y 468.776,Z 882.9,A -85,B 0,C 180,E1 15923.315,E2 15923.315} C_VEL
LIN {X 0,Y 454.466,Z 853.312,A -85,B 0,C 180,E1 15928.299,E2 15928.299} C_VEL
LIN {X 0,Y 439.759,Z 828.774,A -85,B 0,C 180,E1 15933.155,E2 15933.155} C_VEL
LIN {X 0,Y 432.182,Z 816.656,A -85,B 0,C 180,E1 15935.777,E2 15935.777} C_VEL
LIN {X 0,Y 427.784,Z 810.758,A -85,B 0,C 180,E1 15937.237,E2 15937.237} C_VEL
LIN {X 0,Y 427.601,Z 809.06,A -85,B 0,C 180,E1 15937.623,E2 15937.623} C_VEL
LIN {X 0,Y 427.247,Z 809.06,A -85,B 0,C 180,E1 15944.342,E2 15944.342} C_VEL
LIN {X 0,Y 426.878,Z 809.06,A -85,B 0,C 180,E1 15950.74,E2 15950.74} C_VEL
LIN {X 0,Y 426.578,Z 809.06,A -85,B 0,C 180,E1 15957.685,E2 15957.685} C_VEL
LIN {X 0,Y 426.357,Z 809.06,A -85,B 0,C 180,E1 15964.555,E2 15964.555} C_VEL
LIN {X 0,Y 426.279,Z 809.06,A -85,B 0,C 180,E1 15969.657,E2 15969.657} C_VEL
LIN {X 0,Y 426.277,Z 809.06,A -85,B 0,C 180,E1 15975.161,E2 15975.161} C_VEL
LIN {X 0,Y 426.231,Z 809.06,A -85,B 0,C 180,E1 15981.267,E2 15981.267} C_VEL
LIN {X 0,Y 426.44,Z 809.06,A -85,B 0,C 180,E1 15988.272,E2 15988.272} C_VEL
LIN {X 0,Y 426.71,Z 809.06,A -85,B 0,C 180,E1 15994.855,E2 15994.855} C_VEL
LIN {X 0,Y 427.027,Z 809.06,A -85,B 0,C 180,E1 16001.431,E2 16001.431} C_VEL
LIN {X 0,Y 427.357,Z 809.06,A -85,B 0,C 180,E1 16007.753,E2 16007.753} C_VEL
LIN {X 0,Y 427.705,Z 809.06,A -85,B 0,C 180,E1 16013.917,E2 16013.917} C_VEL
LIN {X 0,Y 428.201,Z 809.06,A -85,B 0,C 180,E1 16020.001,E2 16020.001} C_VEL
LIN {X 0,Y 427.724,Z 809.06,A -85,B 0,C 180,E1 16026.084,E2 16026.084} C_VEL
LIN {X 0,Y 427.366,Z 809.06,A -85,B 0,C 180,E1 16032.248,E2 16032.248} C_VEL
LIN {X 0,Y 427.346,Z 809.845,A -85,B 0,C 180,E1 16033.709,E2 16033.709} C_VEL
LIN {X 0,Y 429.975,Z 815.048,A -85,B 0,C 180,E1 16034.631,E2 16034.631} C_VEL
LIN {X 0,Y 432.335,Z 817.763,A -85,B 0,C 180,E1 16035.391,E2 16035.391} C_VEL
LIN {X 0,Y 450.655,Z 843.786,A -85,B 0,C 180,E1 16040.675,E2 16040.675} C_VEL
LIN {X 0,Y 472.214,Z 876.347,A -85,B 0,C 180,E1 16045.985,E2 16045.985} C_VEL
LIN {X 0,Y 492.949,Z 911.05,A -85,B 0,C 180,E1 16050.637,E2 16050.637} C_VEL
LIN {X 0,Y 510.502,Z 946.868,A -85,B 0,C 180,E1 16054.699,E2 16054.699} C_VEL
LIN {X 0,Y 501.507,Z 994.102,A -85,B 0,C 180,E1 16056.451,E2 16056.451} C_VEL
LIN {X 0,Y 490.669,Z 1041.031,A -85,B 0,C 180,E1 16058.97,E2 16058.97} C_VEL
LIN {X 0,Y 478.916,Z 1084.988,A -85,B 0,C 180,E1 16062.133,E2 16062.133} C_VEL
LIN {X 0,Y 465.956,Z 1128.874,A -85,B 0,C 180,E1 16066.321,E2 16066.321} C_VEL
LIN {X 0,Y 454.915,Z 1165.107,A -85,B 0,C 180,E1 16070.858,E2 16070.858} C_VEL
LIN {X 0,Y 444.976,Z 1198.697,A -85,B 0,C 180,E1 16076.255,E2 16076.255} C_VEL
LIN {X 0,Y 437.399,Z 1226.336,A -85,B 0,C 180,E1 16082.032,E2 16082.032} C_VEL
LIN {X 0,Y 432.532,Z 1248.149,A -85,B 0,C 180,E1 16087.97,E2 16087.97} C_VEL
LIN {X 0,Y 429.883,Z 1263.809,A -85,B 0,C 180,E1 16093.66,E2 16093.66} C_VEL
LIN {X 0,Y 428.709,Z 1273.842,A -85,B 0,C 180,E1 16098.814,E2 16098.814} C_VEL
LIN {X 0,Y 428.369,Z 1280.056,A -85,B 0,C 180,E1 16103.917,E2 16103.917} C_VEL
LIN {X 0,Y 428.503,Z 1282.724,A -85,B 0,C 180,E1 16109.992,E2 16109.992} C_VEL
LIN {X 0,Y 428.414,Z 1281.229,A -85,B 0,C 180,E1 16114.037,E2 16114.037} C_VEL
LIN {X 0,Y 428.622,Z 1275.972,A -85,B 0,C 180,E1 16119.222,E2 16119.222} C_VEL
LIN {X 0,Y 429.66,Z 1265.852,A -85,B 0,C 180,E1 16124.773,E2 16124.773} C_VEL
LIN {X 0,Y 427.597,Z 1261.765,A -85,B 0,C 180,E1 16126.415,E2 16126.415} C_VEL
LIN {X 0,Y 423.253,Z 1254.784,A -85,B 0,C 180,E1 16128.854,E2 16128.854} C_VEL
LIN {X 0,Y 423.317,Z 1253.982,A -85,B 0,C 180,E1 16129.133,E2 16129.133} C_VEL
LIN {X 0,Y 427.014,Z 1233.596,A -85,B 0,C 180,E1 16135.118,E2 16135.118} C_VEL
LIN {X 0,Y 432.797,Z 1207.12,A -85,B 0,C 180,E1 16140.984,E2 16140.984} C_VEL
LIN {X 0,Y 440.28,Z 1176.865,A -85,B 0,C 180,E1 16146.178,E2 16146.178} C_VEL
LIN {X 0,Y 449.871,Z 1138.796,A -85,B 0,C 180,E1 16151.24,E2 16151.24} C_VEL
LIN {X 0,Y 460.502,Z 1097.045,A -85,B 0,C 180,E1 16155.564,E2 16155.564} C_VEL
LIN {X 0,Y 472.305,Z 1047.668,A -85,B 0,C 180,E1 16159.476,E2 16159.476} C_VEL
LIN {X 0,Y 484.413,Z 994.297,A -85,B 0,C 180,E1 16162.693,E2 16162.693} C_VEL
LIN {X 0,Y 494.642,Z 947.325,A -85,B 0,C 180,E1 16164.869,E2 16164.869} C_VEL
LIN {X 0,Y 492.541,Z 924.866,A -85,B 0,C 180,E1 16167.529,E2 16167.529} C_VEL
LIN {X 0,Y 493.271,Z 918.339,A -85,B 0,C 180,E1 16168.617,E2 16168.617} C_VEL
LIN {X 0,Y 489.179,Z 932.395,A -85,B 0,C 180,E1 16171.394,E2 16171.394} C_VEL
LIN {X 0,Y 489.163,Z 953.719,A -85,B 0,C 180,E1 16174.866,E2 16174.866} C_VEL
LIN {X 0,Y 476.143,Z 993.276,A -85,B 0,C 180,E1 16178.351,E2 16178.351} C_VEL
LIN {X 0,Y 463.951,Z 1026.659,A -85,B 0,C 180,E1 16182.222,E2 16182.222} C_VEL
LIN {X 0,Y 450.926,Z 1058.932,A -85,B 0,C 180,E1 16187.173,E2 16187.173} C_VEL
LIN {X 0,Y 439.852,Z 1085.298,A -85,B 0,C 180,E1 16192.598,E2 16192.598} C_VEL
LIN {X 0,Y 431.271,Z 1106.889,A -85,B 0,C 180,E1 16198.595,E2 16198.595} C_VEL
LIN {X 0,Y 424.985,Z 1124.361,A -85,B 0,C 180,E1 16205.498,E2 16205.498} C_VEL
LIN {X 0,Y 422.218,Z 1134.473,A -85,B 0,C 180,E1 16211.351,E2 16211.351} C_VEL
LIN {X 0,Y 420.82,Z 1140.306,A -85,B 0,C 180,E1 16216.692,E2 16216.692} C_VEL
LIN {X 0,Y 419.701,Z 1143.362,A -85,B 0,C 180,E1 16223.329,E2 16223.329} C_VEL
LIN {X 0,Y 420.055,Z 1141.752,A -85,B 0,C 180,E1 16230.237,E2 16230.237} C_VEL
LIN {X 0,Y 421.5,Z 1135.492,A -85,B 0,C 180,E1 16236.684,E2 16236.684} C_VEL
LIN {X 0,Y 423.557,Z 1125.57,A -85,B 0,C 180,E1 16242.671,E2 16242.671} C_VEL
LIN {X 0,Y 428.234,Z 1109.371,A -85,B 0,C 180,E1 16249.265,E2 16249.265} C_VEL
LIN {X 0,Y 435.825,Z 1087.078,A -85,B 0,C 180,E1 16255.617,E2 16255.617} C_VEL
LIN {X 0,Y 445.067,Z 1061.812,A -85,B 0,C 180,E1 16260.995,E2 16260.995} C_VEL
LIN {X 0,Y 456.816,Z 1029.46,A -85,B 0,C 180,E1 16266.172,E2 16266.172} C_VEL
LIN {X 0,Y 469.221,Z 993.945,A -85,B 0,C 180,E1 16270.456,E2 16270.456} C_VEL
LIN {X 0,Y 482.359,Z 951.629,A -85,B 0,C 180,E1 16274.313,E2 16274.313} C_VEL
LIN {X 0,Y 483.07,Z 947.8,A -85,B 0,C 180,E1 16274.665,E2 16274.665} C_VEL
LIN {X 0,Y 475.025,Z 918.324,A -85,B 0,C 180,E1 16279.005,E2 16279.005} C_VEL
LIN {X 0,Y 463.171,Z 886.764,A -85,B 0,C 180,E1 16283.921,E2 16283.921} C_VEL
LIN {X 0,Y 449.205,Z 857.814,A -85,B 0,C 180,E1 16288.972,E2 16288.972} C_VEL
LIN {X 0,Y 435.999,Z 835.144,A -85,B 0,C 180,E1 16293.559,E2 16293.559} C_VEL
LIN {X 0,Y 426.926,Z 821.547,A -85,B 0,C 180,E1 16296.741,E2 16296.741} C_VEL
LIN {X 0,Y 422.991,Z 815.495,A -85,B 0,C 180,E1 16298.177,E2 16298.177} C_VEL
LIN {X 0,Y 419.733,Z 810.674,A -85,B 0,C 180,E1 16299.397,E2 16299.397} C_VEL
LIN {X 0,Y 419.58,Z 809.06,A -85,B 0,C 180,E1 16299.596,E2 16299.596} C_VEL
LIN {X 0,Y 419.204,Z 809.06,A -85,B 0,C 180,E1 16306.769,E2 16306.769} C_VEL
LIN {X 0,Y 418.806,Z 809.06,A -85,B 0,C 180,E1 16313.392,E2 16313.392} C_VEL
LIN {X 0,Y 418.591,Z 809.06,A -85,B 0,C 180,E1 16320.366,E2 16320.366} C_VEL
LIN {X 0,Y 418.37,Z 809.06,A -85,B 0,C 180,E1 16327.388,E2 16327.388} C_VEL
LIN {X 0,Y 418.276,Z 809.06,A -85,B 0,C 180,E1 16333.741,E2 16333.741} C_VEL
LIN {X 0,Y 418.262,Z 809.06,A -85,B 0,C 180,E1 16339.44,E2 16339.44} C_VEL
LIN {X 0,Y 418.372,Z 809.06,A -85,B 0,C 180,E1 16346.185,E2 16346.185} C_VEL
LIN {X 0,Y 418.643,Z 809.06,A -85,B 0,C 180,E1 16352.018,E2 16352.018} C_VEL
LIN {X 0,Y 418.928,Z 809.06,A -85,B 0,C 180,E1 16358.859,E2 16358.859} C_VEL
LIN {X 0,Y 419.293,Z 809.06,A -85,B 0,C 180,E1 16365.39,E2 16365.39} C_VEL
LIN {X 0,Y 419.695,Z 809.06,A -85,B 0,C 180,E1 16371.721,E2 16371.721} C_VEL
LIN {X 0,Y 420.097,Z 809.06,A -85,B 0,C 180,E1 16377.94,E2 16377.94} C_VEL
LIN {X 0,Y 420.158,Z 809.06,A -85,B 0,C 180,E1 16382.062,E2 16382.062} C_VEL
LIN {X 0,Y 419.683,Z 809.06,A -85,B 0,C 180,E1 16388.281,E2 16388.281} C_VEL
LIN {X 0,Y 419.468,Z 809.77,A -85,B 0,C 180,E1 16391.494,E2 16391.494} C_VEL
LIN {X 0,Y 422.058,Z 814.94,A -85,B 0,C 180,E1 16392.54,E2 16392.54} C_VEL
LIN {X 0,Y 424.631,Z 817.853,A -85,B 0,C 180,E1 16393.388,E2 16393.388} C_VEL
LIN {X 0,Y 443.565,Z 844.662,A -85,B 0,C 180,E1 16399.205,E2 16399.205} C_VEL
LIN {X 0,Y 466.029,Z 878.352,A -85,B 0,C 180,E1 16404.971,E2 16404.971} C_VEL
LIN {X 0,Y 487.005,Z 913.951,A -85,B 0,C 180,E1 16409.9,E2 16409.9} C_VEL
LIN {X 0,Y 504.708,Z 950.322,A -85,B 0,C 180,E1 16414.149,E2 16414.149} C_VEL
LIN {X 0,Y 495.505,Z 995.844,A -85,B 0,C 180,E1 16415.89,E2 16415.89} C_VEL
LIN {X 0,Y 484.04,Z 1043.763,A -85,B 0,C 180,E1 16418.509,E2 16418.509} C_VEL
LIN {X 0,Y 471.902,Z 1087.309,A -85,B 0,C 180,E1 16421.742,E2 16421.742} C_VEL
LIN {X 0,Y 458.793,Z 1130.309,A -85,B 0,C 180,E1 16425.944,E2 16425.944} C_VEL
LIN {X 0,Y 447.141,Z 1167.202,A -85,B 0,C 180,E1 16430.711,E2 16430.711} C_VEL
LIN {X 0,Y 437.294,Z 1199.341,A -85,B 0,C 180,E1 16436.026,E2 16436.026} C_VEL
LIN {X 0,Y 429.377,Z 1227.291,A -85,B 0,C 180,E1 16442.079,E2 16442.079} C_VEL
LIN {X 0,Y 424.368,Z 1249.455,A -85,B 0,C 180,E1 16448.372,E2 16448.372} C_VEL
LIN {X 0,Y 421.813,Z 1264.832,A -85,B 0,C 180,E1 16454.407,E2 16454.407} C_VEL
LIN {X 0,Y 420.752,Z 1275.445,A -85,B 0,C 180,E1 16460.648,E2 16460.648} C_VEL
LIN {X 0,Y 420.521,Z 1280.217,A -85,B 0,C 180,E1 16465.87,E2 16465.87} C_VEL
LIN {X 0,Y 420.726,Z 1281.448,A -85,B 0,C 180,E1 16469.992,E2 16469.992} C_VEL
LIN {X 0,Y 420.632,Z 1279.919,A -85,B 0,C 180,E1 16474.112,E2 16474.112} C_VEL
LIN {X 0,Y 420.818,Z 1274.568,A -85,B 0,C 180,E1 16479.394,E2 16479.394} C_VEL
LIN {X 0,Y 421.835,Z 1264.987,A -85,B 0,C 180,E1 16484.756,E2 16484.756} C_VEL
LIN {X 0,Y 423.317,Z 1253.982,A -85,B 0,C 180,E1 16489.133,E2 16489.133} C_VEL
LIN {X 0,Y 421.626,Z 1248.952,A -85,B 0,C 180,E1 16490.762,E2 16490.762} C_VEL
LIN {X 0,Y 417.636,Z 1240.654,A -85,B 0,C 180,E1 16493.169,E2 16493.169} C_VEL
LIN {X 0,Y 417.749,Z 1239.698,A -85,B 0,C 180,E1 16493.442,E2 16493.442} C_VEL
LIN {X 0,Y 423.364,Z 1214.289,A -85,B 0,C 180,E1 16499.706,E2 16499.706} C_VEL
LIN {X 0,Y 430.878,Z 1183.947,A -85,B 0,C 180,E1 16505.345,E2 16505.345} C_VEL
LIN {X 0,Y 440.518,Z 1147.066,A -85,B 0,C 180,E1 16510.661,E2 16510.661} C_VEL
LIN {X 0,Y 450.919,Z 1107.385,A -85,B 0,C 180,E1 16515.091,E2 16515.091} C_VEL
LIN {X 0,Y 463.563,Z 1057.85,A -85,B 0,C 180,E1 16519.356,E2 16519.356} C_VEL
LIN {X 0,Y 477.23,Z 1001.143,A -85,B 0,C 180,E1 16523.017,E2 16523.017} C_VEL
LIN {X 0,Y 489.456,Z 950.456,A -85,B 0,C 180,E1 16525.515,E2 16525.515} C_VEL
LIN {X 0,Y 488.962,Z 930.555,A -85,B 0,C 180,E1 16528.017,E2 16528.017} C_VEL
LIN {X 0,Y 489.222,Z 927.52,A -85,B 0,C 180,E1 16528.79,E2 16528.79} C_VEL
LIN {X 0,Y 484.81,Z 941.813,A -85,B 0,C 180,E1 16531.618,E2 16531.618} C_VEL
LIN {X 0,Y 483.977,Z 958.155,A -85,B 0,C 180,E1 16534.317,E2 16534.317} C_VEL
LIN {X 0,Y 469.299,Z 999.935,A -85,B 0,C 180,E1 16538.143,E2 16538.143} C_VEL
LIN {X 0,Y 455.775,Z 1034.427,A -85,B 0,C 180,E1 16542.391,E2 16542.391} C_VEL
LIN {X 0,Y 443.255,Z 1064.107,A -85,B 0,C 180,E1 16547.198,E2 16547.198} C_VEL
LIN {X 0,Y 431.565,Z 1090.605,A -85,B 0,C 180,E1 16552.96,E2 16552.96} C_VEL
LIN {X 0,Y 423.096,Z 1110.851,A -85,B 0,C 180,E1 16558.991,E2 16558.991} C_VEL
LIN {X 0,Y 417.255,Z 1126.775,A -85,B 0,C 180,E1 16565.6,E2 16565.6} C_VEL
LIN {X 0,Y 414.396,Z 1136.445,A -85,B 0,C 180,E1 16571.568,E2 16571.568} C_VEL
LIN {X 0,Y 412.716,Z 1142.539,A -85,B 0,C 180,E1 16577.868,E2 16577.868} C_VEL
LIN {X 0,Y 411.849,Z 1144.71,A -85,B 0,C 180,E1 16583.8,E2 16583.8} C_VEL
LIN {X 0,Y 412.373,Z 1142.634,A -85,B 0,C 180,E1 16590.861,E2 16590.861} C_VEL
LIN {X 0,Y 413.668,Z 1137.15,A -85,B 0,C 180,E1 16596.538,E2 16596.538} C_VEL
LIN {X 0,Y 415.91,Z 1126.878,A -85,B 0,C 180,E1 16602.88,E2 16602.88} C_VEL
LIN {X 0,Y 420.604,Z 1111.271,A -85,B 0,C 180,E1 16609.392,E2 16609.392} C_VEL
LIN {X 0,Y 428.06,Z 1090.04,A -85,B 0,C 180,E1 16615.622,E2 16615.622} C_VEL
LIN {X 0,Y 437.947,Z 1063.958,A -85,B 0,C 180,E1 16621.34,E2 16621.34} C_VEL
LIN {X 0,Y 449.421,Z 1033.178,A -85,B 0,C 180,E1 16626.384,E2 16626.384} C_VEL
LIN {X 0,Y 462.274,Z 997.927,A -85,B 0,C 180,E1 16630.772,E2 16630.772} C_VEL
LIN {X 0,Y 475.197,Z 957.667,A -85,B 0,C 180,E1 16634.55,E2 16634.55} C_VEL
LIN {X 0,Y 476.826,Z 951.042,A -85,B 0,C 180,E1 16635.143,E2 16635.143} C_VEL
LIN {X 0,Y 468.926,Z 921.703,A -85,B 0,C 180,E1 16639.565,E2 16639.565} C_VEL
LIN {X 0,Y 458.04,Z 891.851,A -85,B 0,C 180,E1 16644.328,E2 16644.328} C_VEL
LIN {X 0,Y 444.344,Z 862.844,A -85,B 0,C 180,E1 16649.521,E2 16649.521} C_VEL
LIN {X 0,Y 432.185,Z 841.557,A -85,B 0,C 180,E1 16653.934,E2 16653.934} C_VEL
LIN {X 0,Y 422.554,Z 826.934,A -85,B 0,C 180,E1 16657.45,E2 16657.45} C_VEL
LIN {X 0,Y 419.292,Z 821.884,A -85,B 0,C 180,E1 16658.744,E2 16658.744} C_VEL
LIN {X 0,Y 415.019,Z 815.517,A -85,B 0,C 180,E1 16660.372,E2 16660.372} C_VEL
LIN {X 0,Y 411.688,Z 810.681,A -85,B 0,C 180,E1 16661.722,E2 16661.722} C_VEL
LIN {X 0,Y 411.522,Z 809.06,A -85,B 0,C 180,E1 16661.929,E2 16661.929} C_VEL
LIN {X 0,Y 411.241,Z 809.06,A -85,B 0,C 180,E1 16667.199,E2 16667.199} C_VEL
LIN {X 0,Y 410.848,Z 809.06,A -85,B 0,C 180,E1 16673.873,E2 16673.873} C_VEL
LIN {X 0,Y 410.682,Z 809.06,A -85,B 0,C 180,E1 16678.585,E2 16678.585} C_VEL
LIN {X 0,Y 410.466,Z 809.06,A -85,B 0,C 180,E1 16685.92,E2 16685.92} C_VEL
LIN {X 0,Y 410.311,Z 809.06,A -85,B 0,C 180,E1 16692.566,E2 16692.566} C_VEL
LIN {X 0,Y 410.28,Z 809.06,A -85,B 0,C 180,E1 16698.479,E2 16698.479} C_VEL
LIN {X 0,Y 410.397,Z 809.06,A -85,B 0,C 180,E1 16704.112,E2 16704.112} C_VEL
LIN {X 0,Y 410.681,Z 809.06,A -85,B 0,C 180,E1 16711.427,E2 16711.427} C_VEL
LIN {X 0,Y 410.963,Z 809.06,A -85,B 0,C 180,E1 16718.429,E2 16718.429} C_VEL
LIN {X 0,Y 411.342,Z 809.06,A -85,B 0,C 180,E1 16725.101,E2 16725.101} C_VEL
LIN {X 0,Y 411.766,Z 809.06,A -85,B 0,C 180,E1 16732.29,E2 16732.29} C_VEL
LIN {X 0,Y 412.186,Z 809.06,A -85,B 0,C 180,E1 16737.9,E2 16737.9} C_VEL
LIN {X 0,Y 412.245,Z 809.06,A -85,B 0,C 180,E1 16742.101,E2 16742.101} C_VEL
LIN {X 0,Y 411.685,Z 809.48,A -85,B 0,C 180,E1 16749.174,E2 16749.174} C_VEL
LIN {X 0,Y 413.974,Z 814.688,A -85,B 0,C 180,E1 16750.184,E2 16750.184} C_VEL
LIN {X 0,Y 416.898,Z 817.932,A -85,B 0,C 180,E1 16751.207,E2 16751.207} C_VEL
LIN {X 0,Y 422.9,Z 826.73,A -85,B 0,C 180,E1 16753.368,E2 16753.368} C_VEL
LIN {X 0,Y 436.511,Z 845.555,A -85,B 0,C 180,E1 16757.632,E2 16757.632} C_VEL
LIN {X 0,Y 456.906,Z 875.914,A -85,B 0,C 180,E1 16763.188,E2 16763.188} C_VEL
LIN {X 0,Y 478.955,Z 912.704,A -85,B 0,C 180,E1 16768.629,E2 16768.629} C_VEL
LIN {X 0,Y 498.058,Z 951.648,A -85,B 0,C 180,E1 16773.359,E2 16773.359} C_VEL
LIN {X 0,Y 498.659,Z 954.58,A -85,B 0,C 180,E1 16773.612,E2 16773.612} C_VEL
LIN {X 0,Y 488.682,Z 1001.382,A -85,B 0,C 180,E1 16775.496,E2 16775.496} C_VEL
LIN {X 0,Y 477.409,Z 1046.564,A -85,B 0,C 180,E1 16778.055,E2 16778.055} C_VEL
LIN {X 0,Y 463.844,Z 1093.198,A -85,B 0,C 180,E1 16781.653,E2 16781.653} C_VEL
LIN {X 0,Y 451.291,Z 1132.582,A -85,B 0,C 180,E1 16785.677,E2 16785.677} C_VEL
LIN {X 0,Y 438.99,Z 1170.572,A -85,B 0,C 180,E1 16790.75,E2 16790.75} C_VEL
LIN {X 0,Y 428.805,Z 1202.277,A -85,B 0,C 180,E1 16796.279,E2 16796.279} C_VEL
LIN {X 0,Y 420.977,Z 1229.594,A -85,B 0,C 180,E1 16802.465,E2 16802.465} C_VEL
LIN {X 0,Y 416.261,Z 1250.235,A -85,B 0,C 180,E1 16808.706,E2 16808.706} C_VEL
LIN {X 0,Y 413.778,Z 1265.749,A -85,B 0,C 180,E1 16815.18,E2 16815.18} C_VEL
LIN {X 0,Y 412.878,Z 1275.627,A -85,B 0,C 180,E1 16821.573,E2 16821.573} C_VEL
LIN {X 0,Y 412.776,Z 1279.85,A -85,B 0,C 180,E1 16827.894,E2 16827.894} C_VEL
LIN {X 0,Y 412.978,Z 1279.669,A -85,B 0,C 180,E1 16832.088,E2 16832.088} C_VEL
LIN {X 0,Y 412.937,Z 1274.798,A -85,B 0,C 180,E1 16838.408,E2 16838.408} C_VEL
LIN {X 0,Y 413.887,Z 1265.161,A -85,B 0,C 180,E1 16844.257,E2 16844.257} C_VEL
LIN {X 0,Y 415.911,Z 1250.258,A -85,B 0,C 180,E1 16850.182,E2 16850.182} C_VEL
LIN {X 0,Y 417.749,Z 1239.698,A -85,B 0,C 180,E1 16853.442,E2 16853.442} C_VEL
LIN {X 0,Y 416.446,Z 1233.934,A -85,B 0,C 180,E1 16855.05,E2 16855.05} C_VEL
LIN {X 0,Y 413.05,Z 1224.665,A -85,B 0,C 180,E1 16857.44,E2 16857.44} C_VEL
LIN {X 0,Y 413.207,Z 1223.599,A -85,B 0,C 180,E1 16857.706,E2 16857.706} C_VEL
LIN {X 0,Y 420.172,Z 1195.58,A -85,B 0,C 180,E1 16863.591,E2 16863.591} C_VEL
LIN {X 0,Y 429.13,Z 1162.351,A -85,B 0,C 180,E1 16868.996,E2 16868.996} C_VEL
LIN {X 0,Y 439.687,Z 1123.73,A -85,B 0,C 180,E1 16873.884,E2 16873.884} C_VEL
LIN {X 0,Y 452.48,Z 1076.559,A -85,B 0,C 180,E1 16878.458,E2 16878.458} C_VEL
LIN {X 0,Y 465.023,Z 1028.601,A -85,B 0,C 180,E1 16882.03,E2 16882.03} C_VEL
LIN {X 0,Y 479.261,Z 973.738,A -85,B 0,C 180,E1 16885.177,E2 16885.177} C_VEL
LIN {X 0,Y 484.499,Z 954.307,A -85,B 0,C 180,E1 16886.107,E2 16886.107} C_VEL
LIN {X 0,Y 485.394,Z 937.247,A -85,B 0,C 180,E1 16888.382,E2 16888.382} C_VEL
LIN {X 0,Y 485.593,Z 935.759,A -85,B 0,C 180,E1 16888.753,E2 16888.753} C_VEL
LIN {X 0,Y 480.256,Z 951.246,A -85,B 0,C 180,E1 16891.839,E2 16891.839} C_VEL
LIN {X 0,Y 479.231,Z 961.915,A -85,B 0,C 180,E1 16893.687,E2 16893.687} C_VEL
LIN {X 0,Y 463.251,Z 1004.6,A -85,B 0,C 180,E1 16897.717,E2 16897.717} C_VEL
LIN {X 0,Y 447.64,Z 1042.165,A -85,B 0,C 180,E1 16902.567,E2 16902.567} C_VEL
LIN {X 0,Y 433.45,Z 1073.812,A -85,B 0,C 180,E1 16908.162,E2 16908.162} C_VEL
LIN {X 0,Y 422.477,Z 1097.5,A -85,B 0,C 180,E1 16913.84,E2 16913.84} C_VEL
LIN {X 0,Y 414.351,Z 1116.435,A -85,B 0,C 180,E1 16919.999,E2 16919.999} C_VEL
LIN {X 0,Y 409.078,Z 1130.25,A -85,B 0,C 180,E1 16926.361,E2 16926.361} C_VEL
LIN {X 0,Y 406.186,Z 1139.687,A -85,B 0,C 180,E1 16932.896,E2 16932.896} C_VEL
LIN {X 0,Y 404.575,Z 1145.014,A -85,B 0,C 180,E1 16939.64,E2 16939.64} C_VEL
LIN {X 0,Y 404.039,Z 1145.731,A -85,B 0,C 180,E1 16946.664,E2 16946.664} C_VEL
LIN {X 0,Y 404.916,Z 1142.739,A -85,B 0,C 180,E1 16952.38,E2 16952.38} C_VEL
LIN {X 0,Y 406.696,Z 1135.062,A -85,B 0,C 180,E1 16959.167,E2 16959.167} C_VEL
LIN {X 0,Y 409.669,Z 1123.162,A -85,B 0,C 180,E1 16965.52,E2 16965.52} C_VEL
LIN {X 0,Y 415.903,Z 1104.802,A -85,B 0,C 180,E1 16972.295,E2 16972.295} C_VEL
LIN {X 0,Y 424.207,Z 1082.657,A -85,B 0,C 180,E1 16978.186,E2 16978.186} C_VEL
LIN {X 0,Y 435.081,Z 1054.934,A -85,B 0,C 180,E1 16983.726,E2 16983.726} C_VEL
LIN {X 0,Y 447.513,Z 1022.628,A -85,B 0,C 180,E1 16988.581,E2 16988.581} C_VEL
LIN {X 0,Y 460.998,Z 985.089,A -85,B 0,C 180,E1 16992.851,E2 16992.851} C_VEL
LIN {X 0,Y 470.435,Z 953.867,A -85,B 0,C 180,E1 16995.685,E2 16995.685} C_VEL
LIN {X 0,Y 462.857,Z 924.863,A -85,B 0,C 180,E1 17000.166,E2 17000.166} C_VEL
LIN {X 0,Y 451.946,Z 894.613,A -85,B 0,C 180,E1 17005.153,E2 17005.153} C_VEL
LIN {X 0,Y 438.779,Z 866.175,A -85,B 0,C 180,E1 17010.381,E2 17010.381} C_VEL
LIN {X 0,Y 424.939,Z 842.166,A -85,B 0,C 180,E1 17015.639,E2 17015.639} C_VEL
LIN {X 0,Y 415.618,Z 828.247,A -85,B 0,C 180,E1 17019.223,E2 17019.223} C_VEL
LIN {X 0,Y 411.667,Z 822.208,A -85,B 0,C 180,E1 17020.852,E2 17020.852} C_VEL
LIN {X 0,Y 406.908,Z 815.476,A -85,B 0,C 180,E1 17022.815,E2 17022.815} C_VEL
LIN {X 0,Y 403.62,Z 810.598,A -85,B 0,C 180,E1 17024.272,E2 17024.272} C_VEL
LIN {X 0,Y 403.467,Z 809.06,A -85,B 0,C 180,E1 17024.513,E2 17024.513} C_VEL
LIN {X 0,Y 403.065,Z 809.06,A -85,B 0,C 180,E1 17030.418,E2 17030.418} C_VEL
LIN {X 0,Y 402.82,Z 809.06,A -85,B 0,C 180,E1 17036.762,E2 17036.762} C_VEL
LIN {X 0,Y 402.63,Z 809.06,A -85,B 0,C 180,E1 17041.706,E2 17041.706} C_VEL
LIN {X 0,Y 402.381,Z 809.06,A -85,B 0,C 180,E1 17047.949,E2 17047.949} C_VEL
LIN {X 0,Y 402.411,Z 809.06,A -85,B 0,C 180,E1 17054.487,E2 17054.487} C_VEL
LIN {X 0,Y 402.344,Z 809.06,A -85,B 0,C 180,E1 17060.326,E2 17060.326} C_VEL
LIN {X 0,Y 402.491,Z 809.06,A -85,B 0,C 180,E1 17065.73,E2 17065.73} C_VEL
LIN {X 0,Y 402.674,Z 809.06,A -85,B 0,C 180,E1 17070.804,E2 17070.804} C_VEL
LIN {X 0,Y 402.901,Z 809.06,A -85,B 0,C 180,E1 17075.637,E2 17075.637} C_VEL
LIN {X 0,Y 403.297,Z 809.06,A -85,B 0,C 180,E1 17082.56,E2 17082.56} C_VEL
LIN {X 0,Y 403.672,Z 809.06,A -85,B 0,C 180,E1 17089.214,E2 17089.214} C_VEL
LIN {X 0,Y 404.093,Z 809.06,A -85,B 0,C 180,E1 17095.712,E2 17095.712} C_VEL
LIN {X 0,Y 404.493,Z 809.06,A -85,B 0,C 180,E1 17100.001,E2 17100.001} C_VEL
LIN {X 0,Y 403.942,Z 809.556,A -85,B 0,C 180,E1 17106.664,E2 17106.664} C_VEL
LIN {X 0,Y 406.197,Z 814.661,A -85,B 0,C 180,E1 17107.724,E2 17107.724} C_VEL
LIN {X 0,Y 409.135,Z 817.502,A -85,B 0,C 180,E1 17108.83,E2 17108.83} C_VEL
LIN {X 0,Y 413.31,Z 823.3,A -85,B 0,C 180,E1 17110.467,E2 17110.467} C_VEL
LIN {X 0,Y 430.178,Z 847.631,A -85,B 0,C 180,E1 17116.229,E2 17116.229} C_VEL
LIN {X 0,Y 448.791,Z 874.827,A -85,B 0,C 180,E1 17121.543,E2 17121.543} C_VEL
LIN {X 0,Y 469.804,Z 909.871,A -85,B 0,C 180,E1 17127.02,E2 17127.02} C_VEL
LIN {X 0,Y 487.214,Z 944.003,A -85,B 0,C 180,E1 17131.492,E2 17131.492} C_VEL
LIN {X 0,Y 492.673,Z 957.975,A -85,B 0,C 180,E1 17133.043,E2 17133.043} C_VEL
LIN {X 0,Y 482.34,Z 1004.838,A -85,B 0,C 180,E1 17134.987,E2 17134.987} C_VEL
LIN {X 0,Y 470.767,Z 1049.011,A -85,B 0,C 180,E1 17137.578,E2 17137.578} C_VEL
LIN {X 0,Y 457.459,Z 1093.399,A -85,B 0,C 180,E1 17141.067,E2 17141.067} C_VEL
LIN {X 0,Y 444.631,Z 1132.374,A -85,B 0,C 180,E1 17145.102,E2 17145.102} C_VEL
LIN {X 0,Y 431.652,Z 1171.073,A -85,B 0,C 180,E1 17150.364,E2 17150.364} C_VEL
LIN {X 0,Y 421.027,Z 1203.04,A -85,B 0,C 180,E1 17156.099,E2 17156.099} C_VEL
LIN {X 0,Y 413.265,Z 1229.267,A -85,B 0,C 180,E1 17162.203,E2 17162.203} C_VEL
LIN {X 0,Y 408.591,Z 1248.934,A -85,B 0,C 180,E1 17168.286,E2 17168.286} C_VEL
LIN {X 0,Y 405.977,Z 1264.481,A -85,B 0,C 180,E1 17174.889,E2 17174.889} C_VEL
LIN {X 0,Y 405.052,Z 1274.38,A -85,B 0,C 180,E1 17181.409,E2 17181.409} C_VEL
LIN {X 0,Y 404.968,Z 1278.592,A -85,B 0,C 180,E1 17187.853,E2 17187.853} C_VEL
LIN {X 0,Y 405.192,Z 1278.391,A -85,B 0,C 180,E1 17192.128,E2 17192.128} C_VEL
LIN {X 0,Y 405.148,Z 1273.403,A -85,B 0,C 180,E1 17198.571,E2 17198.571} C_VEL
LIN {X 0,Y 406.131,Z 1263.312,A -85,B 0,C 180,E1 17204.686,E2 17204.686} C_VEL
LIN {X 0,Y 408.497,Z 1246.902,A -85,B 0,C 180,E1 17211.131,E2 17211.131} C_VEL
LIN {X 0,Y 412.522,Z 1226.59,A -85,B 0,C 180,E1 17216.945,E2 17216.945} C_VEL
LIN {X 0,Y 413.207,Z 1223.599,A -85,B 0,C 180,E1 17217.706,E2 17217.706} C_VEL
LIN {X 0,Y 411.505,Z 1214.853,A -85,B 0,C 180,E1 17219.804,E2 17219.804} C_VEL
LIN {X 0,Y 409.936,Z 1205.506,A -85,B 0,C 180,E1 17221.875,E2 17221.875} C_VEL
LIN {X 0,Y 418.514,Z 1173.74,A -85,B 0,C 180,E1 17227.655,E2 17227.655} C_VEL
LIN {X 0,Y 429.058,Z 1136.756,A -85,B 0,C 180,E1 17232.843,E2 17232.843} C_VEL
LIN {X 0,Y 441.796,Z 1091.931,A -85,B 0,C 180,E1 17237.688,E2 17237.688} C_VEL
LIN {X 0,Y 455.518,Z 1042.373,A -85,B 0,C 180,E1 17241.779,E2 17241.779} C_VEL
LIN {X 0,Y 471.326,Z 986.307,A -85,B 0,C 180,E1 17245.325,E2 17245.325} C_VEL
LIN {X 0,Y 479.932,Z 956.545,A -85,B 0,C 180,E1 17246.944,E2 17246.944} C_VEL
LIN {X 0,Y 481.525,Z 944.624,A -85,B 0,C 180,E1 17248.638,E2 17248.638} C_VEL
LIN {X 0,Y 477.302,Z 952.813,A -85,B 0,C 180,E1 17250.614,E2 17250.614} C_VEL
LIN {X 0,Y 474.516,Z 966.42,A -85,B 0,C 180,E1 17253.089,E2 17253.089} C_VEL
LIN {X 0,Y 457.631,Z 1008.307,A -85,B 0,C 180,E1 17257.172,E2 17257.172} C_VEL
LIN {X 0,Y 441.473,Z 1045.189,A -85,B 0,C 180,E1 17262.058,E2 17262.058} C_VEL
LIN {X 0,Y 426.762,Z 1076.512,A -85,B 0,C 180,E1 17267.734,E2 17267.734} C_VEL
LIN {X 0,Y 415.007,Z 1100.679,A -85,B 0,C 180,E1 17273.728,E2 17273.728} C_VEL
LIN {X 0,Y 406.694,Z 1119.145,A -85,B 0,C 180,E1 17279.999,E2 17279.999} C_VEL
LIN {X 0,Y 400.731,Z 1134.386,A -85,B 0,C 180,E1 17287.583,E2 17287.583} C_VEL
LIN {X 0,Y 398.361,Z 1141.654,A -85,B 0,C 180,E1 17293.154,E2 17293.154} C_VEL
LIN {X 0,Y 396.693,Z 1146.514,A -85,B 0,C 180,E1 17300.047,E2 17300.047} C_VEL
LIN {X 0,Y 396.219,Z 1147.374,A -85,B 0,C 180,E1 17304.801,E2 17304.801} C_VEL
LIN {X 0,Y 396.536,Z 1145.847,A -85,B 0,C 180,E1 17309.693,E2 17309.693} C_VEL
LIN {X 0,Y 397.87,Z 1140.932,A -85,B 0,C 180,E1 17315.714,E2 17315.714} C_VEL
LIN {X 0,Y 399.863,Z 1132.436,A -85,B 0,C 180,E1 17321.763,E2 17321.763} C_VEL
LIN {X 0,Y 404.131,Z 1118.279,A -85,B 0,C 180,E1 17328.397,E2 17328.397} C_VEL
LIN {X 0,Y 411.557,Z 1098.35,A -85,B 0,C 180,E1 17334.974,E2 17334.974} C_VEL
LIN {X 0,Y 421.384,Z 1073.67,A -85,B 0,C 180,E1 17340.929,E2 17340.929} C_VEL
LIN {X 0,Y 433.895,Z 1042.737,A -85,B 0,C 180,E1 17346.495,E2 17346.495} C_VEL
LIN {X 0,Y 446.776,Z 1009.416,A -85,B 0,C 180,E1 17350.98,E2 17350.98} C_VEL
LIN {X 0,Y 460.654,Z 969.975,A -85,B 0,C 180,E1 17355.012,E2 17355.012} C_VEL
LIN {X 0,Y 464.297,Z 957.812,A -85,B 0,C 180,E1 17356.066,E2 17356.066} C_VEL
LIN {X 0,Y 456.911,Z 928.391,A -85,B 0,C 180,E1 17360.73,E2 17360.73} C_VEL
LIN {X 0,Y 446.672,Z 899.282,A -85,B 0,C 180,E1 17365.643,E2 17365.643} C_VEL
LIN {X 0,Y 433.995,Z 871.374,A -85,B 0,C 180,E1 17370.942,E2 17370.942} C_VEL
LIN {X 0,Y 421.102,Z 848.544,A -85,B 0,C 180,E1 17376.028,E2 17376.028} C_VEL
LIN {X 0,Y 411.795,Z 834.277,A -85,B 0,C 180,E1 17379.783,E2 17379.783} C_VEL
LIN {X 0,Y 407.798,Z 828.312,A -85,B 0,C 180,E1 17381.5,E2 17381.5} C_VEL
LIN {X 0,Y 403.951,Z 822.502,A -85,B 0,C 180,E1 17383.182,E2 17383.182} C_VEL
LIN {X 0,Y 400.42,Z 816.62,A -85,B 0,C 180,E1 17384.845,E2 17384.845} C_VEL
LIN {X 0,Y 395.809,Z 811.572,A -85,B 0,C 180,E1 17386.903,E2 17386.903} C_VEL
LIN {X 0,Y 395.433,Z 809.06,A -85,B 0,C 180,E1 17387.43,E2 17387.43} C_VEL
LIN {X 0,Y 394.92,Z 809.06,A -85,B 0,C 180,E1 17394.9,E2 17394.9} C_VEL
LIN {X 0,Y 394.752,Z 809.06,A -85,B 0,C 180,E1 17399.853,E2 17399.853} C_VEL
LIN {X 0,Y 394.49,Z 809.06,A -85,B 0,C 180,E1 17406.454,E2 17406.454} C_VEL
LIN {X 0,Y 394.454,Z 809.06,A -85,B 0,C 180,E1 17413.605,E2 17413.605} C_VEL
LIN {X 0,Y 394.445,Z 809.06,A -85,B 0,C 180,E1 17420.024,E2 17420.024} C_VEL
LIN {X 0,Y 394.585,Z 809.06,A -85,B 0,C 180,E1 17427.582,E2 17427.582} C_VEL
LIN {X 0,Y 394.821,Z 809.06,A -85,B 0,C 180,E1 17432.663,E2 17432.663} C_VEL
LIN {X 0,Y 395.236,Z 809.06,A -85,B 0,C 180,E1 17439.876,E2 17439.876} C_VEL
LIN {X 0,Y 395.646,Z 809.06,A -85,B 0,C 180,E1 17446.754,E2 17446.754} C_VEL
LIN {X 0,Y 396.047,Z 809.06,A -85,B 0,C 180,E1 17453.429,E2 17453.429} C_VEL
LIN {X 0,Y 396.589,Z 809.06,A -85,B 0,C 180,E1 17460.001,E2 17460.001} C_VEL
LIN {X 0,Y 396.243,Z 809.467,A -85,B 0,C 180,E1 17463.896,E2 17463.896} C_VEL
LIN {X 0,Y 398.417,Z 814.651,A -85,B 0,C 180,E1 17465.032,E2 17465.032} C_VEL
LIN {X 0,Y 401.469,Z 817.751,A -85,B 0,C 180,E1 17466.348,E2 17466.348} C_VEL
LIN {X 0,Y 405.715,Z 823.344,A -85,B 0,C 180,E1 17468.096,E2 17468.096} C_VEL
LIN {X 0,Y 421.648,Z 846.129,A -85,B 0,C 180,E1 17473.995,E2 17473.995} C_VEL
LIN {X 0,Y 438.711,Z 871.215,A -85,B 0,C 180,E1 17479.278,E2 17479.278} C_VEL
LIN {X 0,Y 458.272,Z 902.67,A -85,B 0,C 180,E1 17484.665,E2 17484.665} C_VEL
LIN {X 0,Y 476.385,Z 936.631,A -85,B 0,C 180,E1 17489.513,E2 17489.513} C_VEL
LIN {X 0,Y 486.972,Z 959.989,A -85,B 0,C 180,E1 17492.417,E2 17492.417} C_VEL
LIN {X 0,Y 476.269,Z 1006.975,A -85,B 0,C 180,E1 17494.409,E2 17494.409} C_VEL
LIN {X 0,Y 463.269,Z 1054.424,A -85,B 0,C 180,E1 17497.294,E2 17497.294} C_VEL
LIN {X 0,Y 450.255,Z 1096.224,A -85,B 0,C 180,E1 17500.702,E2 17500.702} C_VEL
LIN {X 0,Y 435.962,Z 1138.1,A -85,B 0,C 180,E1 17505.244,E2 17505.244} C_VEL
LIN {X 0,Y 424.078,Z 1172.257,A -85,B 0,C 180,E1 17510.096,E2 17510.096} C_VEL
LIN {X 0,Y 412.881,Z 1205.079,A -85,B 0,C 180,E1 17516.183,E2 17516.183} C_VEL
LIN {X 0,Y 405.287,Z 1229.831,A -85,B 0,C 180,E1 17522.213,E2 17522.213} C_VEL
LIN {X 0,Y 400.629,Z 1249.13,A -85,B 0,C 180,E1 17528.414,E2 17528.414} C_VEL
LIN {X 0,Y 398.185,Z 1263.205,A -85,B 0,C 180,E1 17534.586,E2 17534.586} C_VEL
LIN {X 0,Y 397.232,Z 1273.124,A -85,B 0,C 180,E1 17541.239,E2 17541.239} C_VEL
LIN {X 0,Y 397.177,Z 1277.321,A -85,B 0,C 180,E1 17547.811,E2 17547.811} C_VEL
LIN {X 0,Y 397.398,Z 1277.086,A -85,B 0,C 180,E1 17552.17,E2 17552.17} C_VEL
LIN {X 0,Y 397.357,Z 1272.007,A -85,B 0,C 180,E1 17558.74,E2 17558.74} C_VEL
LIN {X 0,Y 398.314,Z 1262.221,A -85,B 0,C 180,E1 17564.775,E2 17564.775} C_VEL
LIN {X 0,Y 400.555,Z 1246.896,A -85,B 0,C 180,E1 17570.991,E2 17570.991} C_VEL
LIN {X 0,Y 404.778,Z 1225.815,A -85,B 0,C 180,E1 17577.203,E2 17577.203} C_VEL
LIN {X 0,Y 409.936,Z 1205.506,A -85,B 0,C 180,E1 17581.875,E2 17581.875} C_VEL
LIN {X 0,Y 408.551,Z 1195.946,A -85,B 0,C 180,E1 17583.922,E2 17583.922} C_VEL
LIN {X 0,Y 407.657,Z 1185.872,A -85,B 0,C 180,E1 17585.94,E2 17585.94} C_VEL
LIN {X 0,Y 417.371,Z 1152.422,A -85,B 0,C 180,E1 17591.263,E2 17591.263} C_VEL
LIN {X 0,Y 429.936,Z 1109.888,A -85,B 0,C 180,E1 17596.476,E2 17596.476} C_VEL
LIN {X 0,Y 443.77,Z 1063.072,A -85,B 0,C 180,E1 17600.885,E2 17600.885} C_VEL
LIN {X 0,Y 462.561,Z 1000.235,A -85,B 0,C 180,E1 17605.352,E2 17605.352} C_VEL
LIN {X 0,Y 475.902,Z 959.934,A -85,B 0,C 180,E1 17607.701,E2 17607.701} C_VEL
LIN {X 0,Y 477.313,Z 953.201,A -85,B 0,C 180,E1 17608.718,E2 17608.718} C_VEL
LIN {X 0,Y 471.76,Z 964.291,A -85,B 0,C 180,E1 17611.286,E2 17611.286} C_VEL
LIN {X 0,Y 470.042,Z 970.958,A -85,B 0,C 180,E1 17612.469,E2 17612.469} C_VEL
LIN {X 0,Y 452.133,Z 1012.121,A -85,B 0,C 180,E1 17616.618,E2 17616.618} C_VEL
LIN {X 0,Y 436.078,Z 1046.859,A -85,B 0,C 180,E1 17621.306,E2 17621.306} C_VEL
LIN {X 0,Y 420.719,Z 1077.976,A -85,B 0,C 180,E1 17627.028,E2 17627.028} C_VEL
LIN {X 0,Y 408.386,Z 1102.113,A -85,B 0,C 180,E1 17633.093,E2 17633.093} C_VEL
LIN {X 0,Y 399.719,Z 1120.376,A -85,B 0,C 180,E1 17639.383,E2 17639.383} C_VEL
LIN {X 0,Y 393.537,Z 1134.816,A -85,B 0,C 180,E1 17646.613,E2 17646.613} C_VEL
LIN {X 0,Y 390.564,Z 1143.582,A -85,B 0,C 180,E1 17653.421,E2 17653.421} C_VEL
LIN {X 0,Y 388.826,Z 1148.006,A -85,B 0,C 180,E1 17660.471,E2 17660.471} C_VEL
LIN {X 0,Y 388.519,Z 1148.049,A -85,B 0,C 180,E1 17667.819,E2 17667.819} C_VEL
LIN {X 0,Y 389.681,Z 1144.144,A -85,B 0,C 180,E1 17673.96,E2 17673.96} C_VEL
LIN {X 0,Y 391.492,Z 1136.632,A -85,B 0,C 180,E1 17680.141,E2 17680.141} C_VEL
LIN {X 0,Y 395.276,Z 1123.414,A -85,B 0,C 180,E1 17687.122,E2 17687.122} C_VEL
LIN {X 0,Y 401.678,Z 1106.509,A -85,B 0,C 180,E1 17693.375,E2 17693.375} C_VEL
LIN {X 0,Y 410.948,Z 1083.402,A -85,B 0,C 180,E1 17699.577,E2 17699.577} C_VEL
LIN {X 0,Y 422.804,Z 1055.259,A -85,B 0,C 180,E1 17705.243,E2 17705.243} C_VEL
LIN {X 0,Y 436.264,Z 1021.907,A -85,B 0,C 180,E1 17710.218,E2 17710.218} C_VEL
LIN {X 0,Y 450.333,Z 984.567,A -85,B 0,C 180,E1 17714.437,E2 17714.437} C_VEL
LIN {X 0,Y 457.918,Z 960.576,A -85,B 0,C 180,E1 17716.653,E2 17716.653} C_VEL
LIN {X 0,Y 450.89,Z 931.713,A -85,B 0,C 180,E1 17721.334,E2 17721.334} C_VEL
LIN {X 0,Y 441.036,Z 902.968,A -85,B 0,C 180,E1 17726.32,E2 17726.32} C_VEL
LIN {X 0,Y 429.49,Z 877.004,A -85,B 0,C 180,E1 17731.388,E2 17731.388} C_VEL
LIN {X 0,Y 417.244,Z 854.824,A -85,B 0,C 180,E1 17736.441,E2 17736.441} C_VEL
LIN {X 0,Y 405.62,Z 836.213,A -85,B 0,C 180,E1 17741.441,E2 17741.441} C_VEL
LIN {X 0,Y 399.705,Z 828.108,A -85,B 0,C 180,E1 17744.082,E2 17744.082} C_VEL
LIN {X 0,Y 396.34,Z 822.889,A -85,B 0,C 180,E1 17745.697,E2 17745.697} C_VEL
LIN {X 0,Y 392.616,Z 817.243,A -85,B 0,C 180,E1 17747.563,E2 17747.563} C_VEL
LIN {X 0,Y 387.676,Z 811.462,A -85,B 0,C 180,E1 17750.07,E2 17750.07} C_VEL
LIN {X 0,Y 387.228,Z 809.06,A -85,B 0,C 180,E1 17750.57,E2 17750.57} C_VEL
LIN {X 0,Y 386.887,Z 809.06,A -85,B 0,C 180,E1 17757.959,E2 17757.959} C_VEL
LIN {X 0,Y 386.606,Z 809.06,A -85,B 0,C 180,E1 17765.904,E2 17765.904} C_VEL
LIN {X 0,Y 386.456,Z 809.06,A -85,B 0,C 180,E1 17772.025,E2 17772.025} C_VEL
LIN {X 0,Y 386.438,Z 809.06,A -85,B 0,C 180,E1 17778.341,E2 17778.341} C_VEL
LIN {X 0,Y 386.587,Z 809.06,A -85,B 0,C 180,E1 17785.183,E2 17785.183} C_VEL
LIN {X 0,Y 386.887,Z 809.06,A -85,B 0,C 180,E1 17792.054,E2 17792.054} C_VEL
LIN {X 0,Y 387.271,Z 809.06,A -85,B 0,C 180,E1 17799.486,E2 17799.486} C_VEL
LIN {X 0,Y 387.729,Z 809.06,A -85,B 0,C 180,E1 17807.02,E2 17807.02} C_VEL
LIN {X 0,Y 388.137,Z 809.06,A -85,B 0,C 180,E1 17813.294,E2 17813.294} C_VEL
LIN {X 0,Y 388.687,Z 809.06,A -85,B 0,C 180,E1 17820.001,E2 17820.001} C_VEL
LIN {X 0,Y 388.564,Z 809.432,A -85,B 0,C 180,E1 17820.836,E2 17820.836} C_VEL
LIN {X 0,Y 390.711,Z 814.484,A -85,B 0,C 180,E1 17822.079,E2 17822.079} C_VEL
LIN {X 0,Y 393.844,Z 817.716,A -85,B 0,C 180,E1 17823.588,E2 17823.588} C_VEL
LIN {X 0,Y 397.768,Z 823.264,A -85,B 0,C 180,E1 17825.382,E2 17825.382} C_VEL
LIN {X 0,Y 405.375,Z 834.304,A -85,B 0,C 180,E1 17828.643,E2 17828.643} C_VEL
LIN {X 0,Y 415.93,Z 848.953,A -85,B 0,C 180,E1 17832.591,E2 17832.591} C_VEL
LIN {X 0,Y 431.943,Z 872.212,A -85,B 0,C 180,E1 17837.808,E2 17837.808} C_VEL
LIN {X 0,Y 451.434,Z 903.661,A -85,B 0,C 180,E1 17843.481,E2 17843.481} C_VEL
LIN {X 0,Y 470.32,Z 939.163,A -85,B 0,C 180,E1 17848.745,E2 17848.745} C_VEL
LIN {X 0,Y 480.904,Z 964.323,A -85,B 0,C 180,E1 17851.868,E2 17851.868} C_VEL
LIN {X 0,Y 470.474,Z 1007.969,A -85,B 0,C 180,E1 17853.772,E2 17853.772} C_VEL
LIN {X 0,Y 456.775,Z 1056.489,A -85,B 0,C 180,E1 17856.777,E2 17856.777} C_VEL
LIN {X 0,Y 443.606,Z 1097.246,A -85,B 0,C 180,E1 17860.174,E2 17860.174} C_VEL
LIN {X 0,Y 428.865,Z 1139.073,A -85,B 0,C 180,E1 17864.802,E2 17864.802} C_VEL
LIN {X 0,Y 416.054,Z 1174.647,A -85,B 0,C 180,E1 17870.029,E2 17870.029} C_VEL
LIN {X 0,Y 405.133,Z 1205.664,A -85,B 0,C 180,E1 17875.971,E2 17875.971} C_VEL
LIN {X 0,Y 397.312,Z 1230.397,A -85,B 0,C 180,E1 17882.23,E2 17882.23} C_VEL
LIN {X 0,Y 392.323,Z 1250.781,A -85,B 0,C 180,E1 17889.119,E2 17889.119} C_VEL
LIN {X 0,Y 390.075,Z 1264.316,A -85,B 0,C 180,E1 17895.56,E2 17895.56} C_VEL
LIN {X 0,Y 389.412,Z 1271.867,A -85,B 0,C 180,E1 17901.062,E2 17901.062} C_VEL
LIN {X 0,Y 389.365,Z 1276.058,A -85,B 0,C 180,E1 17907.767,E2 17907.767} C_VEL
LIN {X 0,Y 389.614,Z 1275.777,A -85,B 0,C 180,E1 17912.214,E2 17912.214} C_VEL
LIN {X 0,Y 389.542,Z 1270.606,A -85,B 0,C 180,E1 17918.917,E2 17918.917} C_VEL
LIN {X 0,Y 390.54,Z 1260.726,A -85,B 0,C 180,E1 17925.066,E2 17925.066} C_VEL
LIN {X 0,Y 392.871,Z 1245.21,A -85,B 0,C 180,E1 17931.422,E2 17931.422} C_VEL
LIN {X 0,Y 397.335,Z 1223.968,A -85,B 0,C 180,E1 17937.752,E2 17937.752} C_VEL
LIN {X 0,Y 404.298,Z 1197.689,A -85,B 0,C 180,E1 17943.715,E2 17943.715} C_VEL
LIN {X 0,Y 407.657,Z 1185.872,A -85,B 0,C 180,E1 17945.94,E2 17945.94} C_VEL
LIN {X 0,Y 406.985,Z 1175.601,A -85,B 0,C 180,E1 17947.936,E2 17947.936} C_VEL
LIN {X 0,Y 406.467,Z 1164.741,A -85,B 0,C 180,E1 17949.88,E2 17949.88} C_VEL
LIN {X 0,Y 418.912,Z 1124.097,A -85,B 0,C 180,E1 17955.449,E2 17955.449} C_VEL
LIN {X 0,Y 432.955,Z 1079.336,A -85,B 0,C 180,E1 17960.145,E2 17960.145} C_VEL
LIN {X 0,Y 451.545,Z 1020.508,A -85,B 0,C 180,E1 17964.859,E2 17964.859} C_VEL
LIN {X 0,Y 472.134,Z 964.262,A -85,B 0,C 180,E1 17968.364,E2 17968.364} C_VEL
LIN {X 0,Y 472.723,Z 962.061,A -85,B 0,C 180,E1 17968.707,E2 17968.707} C_VEL
LIN {X 0,Y 470.39,Z 965.139,A -85,B 0,C 180,E1 17969.738,E2 17969.738} C_VEL
LIN {X 0,Y 465.842,Z 975.706,A -85,B 0,C 180,E1 17971.838,E2 17971.838} C_VEL
LIN {X 0,Y 445.874,Z 1017.882,A -85,B 0,C 180,E1 17976.269,E2 17976.269} C_VEL
LIN {X 0,Y 429.323,Z 1051.431,A -85,B 0,C 180,E1 17981,E2 17981} C_VEL
LIN {X 0,Y 414.191,Z 1080.724,A -85,B 0,C 180,E1 17986.551,E2 17986.551} C_VEL
LIN {X 0,Y 400.945,Z 1105.351,A -85,B 0,C 180,E1 17992.964,E2 17992.964} C_VEL
LIN {X 0,Y 391.911,Z 1123.314,A -85,B 0,C 180,E1 17999.492,E2 17999.492} C_VEL
LIN {X 0,Y 385.789,Z 1137.11,A -85,B 0,C 180,E1 18006.747,E2 18006.747} C_VEL
LIN {X 0,Y 382.72,Z 1145.397,A -85,B 0,C 180,E1 18013.702,E2 18013.702} C_VEL
LIN {X 0,Y 381.437,Z 1148.644,A -85,B 0,C 180,E1 18018.475,E2 18018.475} C_VEL
LIN {X 0,Y 380.601,Z 1149.745,A -85,B 0,C 180,E1 18025.893,E2 18025.893} C_VEL
LIN {X 0,Y 381.397,Z 1146.979,A -85,B 0,C 180,E1 18032.018,E2 18032.018} C_VEL
LIN {X 0,Y 383.358,Z 1139.652,A -85,B 0,C 180,E1 18039.096,E2 18039.096} C_VEL
LIN {X 0,Y 386.564,Z 1128.48,A -85,B 0,C 180,E1 18045.732,E2 18045.732} C_VEL
LIN {X 0,Y 393.008,Z 1110.947,A -85,B 0,C 180,E1 18052.721,E2 18052.721} C_VEL
LIN {X 0,Y 401.99,Z 1089.567,A -85,B 0,C 180,E1 18058.932,E2 18058.932} C_VEL
LIN {X 0,Y 413.625,Z 1062.417,A -85,B 0,C 180,E1 18064.74,E2 18064.74} C_VEL
LIN {X 0,Y 427.621,Z 1029.45,A -85,B 0,C 180,E1 18070.024,E2 18070.024} C_VEL
LIN {X 0,Y 442.582,Z 990.968,A -85,B 0,C 180,E1 18074.581,E2 18074.581} C_VEL
LIN {X 0,Y 451.729,Z 964.157,A -85,B 0,C 180,E1 18077.103,E2 18077.103} C_VEL
LIN {X 0,Y 445.307,Z 936.432,A -85,B 0,C 180,E1 18081.716,E2 18081.716} C_VEL
LIN {X 0,Y 435.948,Z 908,A -85,B 0,C 180,E1 18086.775,E2 18086.775} C_VEL
LIN {X 0,Y 424.372,Z 881.532,A -85,B 0,C 180,E1 18092.049,E2 18092.049} C_VEL
LIN {X 0,Y 411.622,Z 857.864,A -85,B 0,C 180,E1 18097.648,E2 18097.648} C_VEL
LIN {X 0,Y 400.898,Z 841.228,A -85,B 0,C 180,E1 18102.418,E2 18102.418} C_VEL
LIN {X 0,Y 393.137,Z 829.65,A -85,B 0,C 180,E1 18106.199,E2 18106.199} C_VEL
LIN {X 0,Y 388.36,Z 822.923,A -85,B 0,C 180,E1 18108.652,E2 18108.652} C_VEL
LIN {X 0,Y 384.692,Z 817.363,A -85,B 0,C 180,E1 18110.712,E2 18110.712} C_VEL
LIN {X 0,Y 379.379,Z 811.251,A -85,B 0,C 180,E1 18113.734,E2 18113.734} C_VEL
LIN {X 0,Y 379.022,Z 809.06,A -85,B 0,C 180,E1 18114.285,E2 18114.285} C_VEL
LIN {X 0,Y 378.762,Z 809.06,A -85,B 0,C 180,E1 18121.251,E2 18121.251} C_VEL
LIN {X 0,Y 378.576,Z 809.06,A -85,B 0,C 180,E1 18127.038,E2 18127.038} C_VEL
LIN {X 0,Y 378.467,Z 809.06,A -85,B 0,C 180,E1 18134.06,E2 18134.06} C_VEL
LIN {X 0,Y 378.453,Z 809.06,A -85,B 0,C 180,E1 18140.298,E2 18140.298} C_VEL
LIN {X 0,Y 378.731,Z 809.06,A -85,B 0,C 180,E1 18146.931,E2 18146.931} C_VEL
LIN {X 0,Y 379.034,Z 809.06,A -85,B 0,C 180,E1 18153.992,E2 18153.992} C_VEL
LIN {X 0,Y 379.421,Z 809.06,A -85,B 0,C 180,E1 18161.423,E2 18161.423} C_VEL
LIN {X 0,Y 379.902,Z 809.06,A -85,B 0,C 180,E1 18168.53,E2 18168.53} C_VEL
LIN {X 0,Y 380.339,Z 809.06,A -85,B 0,C 180,E1 18175.444,E2 18175.444} C_VEL
LIN {X 0,Y 380.513,Z 809.543,A -85,B 0,C 180,E1 18177.227,E2 18177.227} C_VEL
LIN {X 0,Y 383.115,Z 814.816,A -85,B 0,C 180,E1 18178.871,E2 18178.871} C_VEL
LIN {X 0,Y 386.193,Z 817.435,A -85,B 0,C 180,E1 18180.491,E2 18180.491} C_VEL
LIN {X 0,Y 389.983,Z 823.137,A -85,B 0,C 180,E1 18182.461,E2 18182.461} C_VEL
LIN {X 0,Y 391.952,Z 826.171,A -85,B 0,C 180,E1 18183.482,E2 18183.482} C_VEL
LIN {X 0,Y 397.497,Z 833.886,A -85,B 0,C 180,E1 18186.018,E2 18186.018} C_VEL
LIN {X 0,Y 407.272,Z 847.392,A -85,B 0,C 180,E1 18190.016,E2 18190.016} C_VEL
LIN {X 0,Y 423.957,Z 871.311,A -85,B 0,C 180,E1 18195.867,E2 18195.867} C_VEL
LIN {X 0,Y 443.033,Z 902.1,A -85,B 0,C 180,E1 18201.772,E2 18201.772} C_VEL
LIN {X 0,Y 461.571,Z 936.35,A -85,B 0,C 180,E1 18207.195,E2 18207.195} C_VEL
LIN {X 0,Y 475.126,Z 966.428,A -85,B 0,C 180,E1 18211.195,E2 18211.195} C_VEL
LIN {X 0,Y 463.181,Z 1014.574,A -85,B 0,C 180,E1 18213.428,E2 18213.428} C_VEL
LIN {X 0,Y 449.62,Z 1060.617,A -85,B 0,C 180,E1 18216.4,E2 18216.4} C_VEL
LIN {X 0,Y 434.623,Z 1104.794,A -85,B 0,C 180,E1 18220.283,E2 18220.283} C_VEL
LIN {X 0,Y 421.316,Z 1141.354,A -85,B 0,C 180,E1 18224.524,E2 18224.524} C_VEL
LIN {X 0,Y 407.238,Z 1178.923,A -85,B 0,C 180,E1 18230.288,E2 18230.288} C_VEL
LIN {X 0,Y 396.924,Z 1207.49,A -85,B 0,C 180,E1 18236.066,E2 18236.066} C_VEL
LIN {X 0,Y 388.72,Z 1233.254,A -85,B 0,C 180,E1 18242.946,E2 18242.946} C_VEL
LIN {X 0,Y 384.131,Z 1251.952,A -85,B 0,C 180,E1 18249.733,E2 18249.733} C_VEL
LIN {X 0,Y 382.088,Z 1264.562,A -85,B 0,C 180,E1 18256.264,E2 18256.264} C_VEL
LIN {X 0,Y 381.451,Z 1271.61,A -85,B 0,C 180,E1 18262.015,E2 18262.015} C_VEL
LIN {X 0,Y 381.572,Z 1274.796,A -85,B 0,C 180,E1 18267.721,E2 18267.721} C_VEL
LIN {X 0,Y 381.819,Z 1274.482,A -85,B 0,C 180,E1 18272.259,E2 18272.259} C_VEL
LIN {X 0,Y 381.751,Z 1269.21,A -85,B 0,C 180,E1 18279.1,E2 18279.1} C_VEL
LIN {X 0,Y 382.743,Z 1258.965,A -85,B 0,C 180,E1 18285.488,E2 18285.488} C_VEL
LIN {X 0,Y 385.198,Z 1243.541,A -85,B 0,C 180,E1 18291.87,E2 18291.87} C_VEL
LIN {X 0,Y 389.905,Z 1222.291,A -85,B 0,C 180,E1 18298.295,E2 18298.295} C_VEL
LIN {X 0,Y 397.29,Z 1195.341,A -85,B 0,C 180,E1 18304.464,E2 18304.464} C_VEL
LIN {X 0,Y 406.467,Z 1164.741,A -85,B 0,C 180,E1 18309.88,E2 18309.88} C_VEL
LIN {X 0,Y 406.176,Z 1153.666,A -85,B 0,C 180,E1 18311.798,E2 18311.798} C_VEL
LIN {X 0,Y 405.866,Z 1143.791,A -85,B 0,C 180,E1 18313.463,E2 18313.463} C_VEL
LIN {X 0,Y 406.305,Z 1142.254,A -85,B 0,C 180,E1 18313.677,E2 18313.677} C_VEL
LIN {X 0,Y 420.619,Z 1098.51,A -85,B 0,C 180,E1 18318.961,E2 18318.961} C_VEL
LIN {X 0,Y 439.255,Z 1042.67,A -85,B 0,C 180,E1 18324.035,E2 18324.035} C_VEL
LIN {X 0,Y 458.894,Z 990.529,A -85,B 0,C 180,E1 18327.747,E2 18327.747} C_VEL
LIN {X 0,Y 467.195,Z 972.052,A -85,B 0,C 180,E1 18328.88,E2 18328.88} C_VEL
LIN {X 0,Y 467.636,Z 970.726,A -85,B 0,C 180,E1 18329.139,E2 18329.139} C_VEL
LIN {X 0,Y 463.03,Z 978.598,A -85,B 0,C 180,E1 18330.967,E2 18330.967} C_VEL
LIN {X 0,Y 439.662,Z 1023.777,A -85,B 0,C 180,E1 18335.913,E2 18335.913} C_VEL
LIN {X 0,Y 421.894,Z 1057.462,A -85,B 0,C 180,E1 18340.924,E2 18340.924} C_VEL
LIN {X 0,Y 407.037,Z 1084.532,A -85,B 0,C 180,E1 18346.31,E2 18346.31} C_VEL
LIN {X 0,Y 393.534,Z 1108.602,A -85,B 0,C 180,E1 18352.831,E2 18352.831} C_VEL
LIN {X 0,Y 383.65,Z 1127.127,A -85,B 0,C 180,E1 18359.999,E2 18359.999} C_VEL
LIN {X 0,Y 378.035,Z 1139.419,A -85,B 0,C 180,E1 18366.886,E2 18366.886} C_VEL
LIN {X 0,Y 374.854,Z 1147.226,A -85,B 0,C 180,E1 18373.995,E2 18373.995} C_VEL
LIN {X 0,Y 373.569,Z 1150.311,A -85,B 0,C 180,E1 18378.879,E2 18378.879} C_VEL
LIN {X 0,Y 372.785,Z 1150.905,A -85,B 0,C 180,E1 18386.477,E2 18386.477} C_VEL
LIN {X 0,Y 373.842,Z 1147.514,A -85,B 0,C 180,E1 18393.073,E2 18393.073} C_VEL
LIN {X 0,Y 375.913,Z 1139.99,A -85,B 0,C 180,E1 18400.024,E2 18400.024} C_VEL
LIN {X 0,Y 380.012,Z 1126.585,A -85,B 0,C 180,E1 18407.483,E2 18407.483} C_VEL
LIN {X 0,Y 387.447,Z 1108.386,A -85,B 0,C 180,E1 18414.445,E2 18414.445} C_VEL
LIN {X 0,Y 397.634,Z 1084.676,A -85,B 0,C 180,E1 18420.924,E2 18420.924} C_VEL
LIN {X 0,Y 410.522,Z 1055.864,A -85,B 0,C 180,E1 18426.755,E2 18426.755} C_VEL
LIN {X 0,Y 425.058,Z 1021.887,A -85,B 0,C 180,E1 18431.832,E2 18431.832} C_VEL
LIN {X 0,Y 439.261,Z 985.628,A -85,B 0,C 180,E1 18435.92,E2 18435.92} C_VEL
LIN {X 0,Y 445.489,Z 967.205,A -85,B 0,C 180,E1 18437.652,E2 18437.652} C_VEL
LIN {X 0,Y 439.328,Z 939.769,A -85,B 0,C 180,E1 18442.349,E2 18442.349} C_VEL
LIN {X 0,Y 430.232,Z 911.556,A -85,B 0,C 180,E1 18447.492,E2 18447.492} C_VEL
LIN {X 0,Y 418.506,Z 884.282,A -85,B 0,C 180,E1 18453.113,E2 18453.113} C_VEL
LIN {X 0,Y 405.579,Z 860.672,A -85,B 0,C 180,E1 18459.026,E2 18459.026} C_VEL
LIN {X 0,Y 394.078,Z 842.505,A -85,B 0,C 180,E1 18464.539,E2 18464.539} C_VEL
LIN {X 0,Y 389.311,Z 835.784,A -85,B 0,C 180,E1 18466.933,E2 18466.933} C_VEL
LIN {X 0,Y 385.638,Z 830.151,A -85,B 0,C 180,E1 18468.99,E2 18468.99} C_VEL
LIN {X 0,Y 380.814,Z 823.342,A -85,B 0,C 180,E1 18471.756,E2 18471.756} C_VEL
LIN {X 0,Y 376.844,Z 817.971,A -85,B 0,C 180,E1 18474.224,E2 18474.224} C_VEL
LIN {X 0,Y 374.818,Z 815.77,A -85,B 0,C 180,E1 18475.527,E2 18475.527} C_VEL
LIN {X 0,Y 371.136,Z 810.694,A -85,B 0,C 180,E1 18478.093,E2 18478.093} C_VEL
LIN {X 0,Y 370.978,Z 809.06,A -85,B 0,C 180,E1 18478.604,E2 18478.604} C_VEL
LIN {X 0,Y 370.642,Z 809.06,A -85,B 0,C 180,E1 18485.381,E2 18485.381} C_VEL
LIN {X 0,Y 370.594,Z 809.06,A -85,B 0,C 180,E1 18492.787,E2 18492.787} C_VEL
LIN {X 0,Y 370.567,Z 809.06,A -85,B 0,C 180,E1 18499.278,E2 18499.278} C_VEL
LIN {X 0,Y 370.627,Z 809.06,A -85,B 0,C 180,E1 18505.198,E2 18505.198} C_VEL
LIN {X 0,Y 370.896,Z 809.06,A -85,B 0,C 180,E1 18510.735,E2 18510.735} C_VEL
LIN {X 0,Y 371.18,Z 809.06,A -85,B 0,C 180,E1 18515.98,E2 18515.98} C_VEL
LIN {X 0,Y 371.616,Z 809.06,A -85,B 0,C 180,E1 18523.465,E2 18523.465} C_VEL
LIN {X 0,Y 372.121,Z 809.06,A -85,B 0,C 180,E1 18530.654,E2 18530.654} C_VEL
LIN {X 0,Y 372.316,Z 809.747,A -85,B 0,C 180,E1 18532.935,E2 18532.935} C_VEL
LIN {X 0,Y 375.075,Z 815.005,A -85,B 0,C 180,E1 18534.995,E2 18534.995} C_VEL
LIN {X 0,Y 378.361,Z 817.607,A -85,B 0,C 180,E1 18536.944,E2 18536.944} C_VEL
LIN {X 0,Y 382.12,Z 823.056,A -85,B 0,C 180,E1 18539.151,E2 18539.151} C_VEL
LIN {X 0,Y 384.112,Z 825.383,A -85,B 0,C 180,E1 18540.257,E2 18540.257} C_VEL
LIN {X 0,Y 389.919,Z 833.853,A -85,B 0,C 180,E1 18543.264,E2 18543.264} C_VEL
LIN {X 0,Y 399.415,Z 846.763,A -85,B 0,C 180,E1 18547.508,E2 18547.508} C_VEL
LIN {X 0,Y 414.473,Z 868.652,A -85,B 0,C 180,E1 18553.305,E2 18553.305} C_VEL
LIN {X 0,Y 430.487,Z 893.641,A -85,B 0,C 180,E1 18558.672,E2 18558.672} C_VEL
LIN {X 0,Y 448.227,Z 924.91,A -85,B 0,C 180,E1 18564.172,E2 18564.172} C_VEL
LIN {X 0,Y 463.457,Z 956.265,A -85,B 0,C 180,E1 18568.811,E2 18568.811} C_VEL
LIN {X 0,Y 469.188,Z 969.732,A -85,B 0,C 180,E1 18570.603,E2 18570.603} C_VEL
LIN {X 0,Y 455.967,Z 1020.728,A -85,B 0,C 180,E1 18573.049,E2 18573.049} C_VEL
LIN {X 0,Y 441.995,Z 1065.762,A -85,B 0,C 180,E1 18576.118,E2 18576.118} C_VEL
LIN {X 0,Y 426.884,Z 1108.74,A -85,B 0,C 180,E1 18580.039,E2 18580.039} C_VEL
LIN {X 0,Y 411.917,Z 1148.063,A -85,B 0,C 180,E1 18584.875,E2 18584.875} C_VEL
LIN {X 0,Y 399.081,Z 1181.286,A -85,B 0,C 180,E1 18590.243,E2 18590.243} C_VEL
LIN {X 0,Y 388.049,Z 1210.98,A -85,B 0,C 180,E1 18596.585,E2 18596.585} C_VEL
LIN {X 0,Y 380.722,Z 1233.765,A -85,B 0,C 180,E1 18602.978,E2 18602.978} C_VEL
LIN {X 0,Y 376.252,Z 1251.484,A -85,B 0,C 180,E1 18609.693,E2 18609.693} C_VEL
LIN {X 0,Y 374.288,Z 1263.279,A -85,B 0,C 180,E1 18615.972,E2 18615.972} C_VEL
LIN {X 0,Y 373.762,Z 1269.324,A -85,B 0,C 180,E1 18620.684,E2 18620.684} C_VEL
LIN {X 0,Y 373.786,Z 1273.518,A -85,B 0,C 180,E1 18627.674,E2 18627.674} C_VEL
LIN {X 0,Y 374.012,Z 1273.162,A -85,B 0,C 180,E1 18632.306,E2 18632.306} C_VEL
LIN {X 0,Y 373.917,Z 1268.689,A -85,B 0,C 180,E1 18638.45,E2 18638.45} C_VEL
LIN {X 0,Y 374.769,Z 1259.721,A -85,B 0,C 180,E1 18644.615,E2 18644.615} C_VEL
LIN {X 0,Y 376.946,Z 1245.231,A -85,B 0,C 180,E1 18651.138,E2 18651.138} C_VEL
LIN {X 0,Y 381.387,Z 1224.842,A -85,B 0,C 180,E1 18657.708,E2 18657.708} C_VEL
LIN {X 0,Y 388.579,Z 1198.992,A -85,B 0,C 180,E1 18663.975,E2 18663.975} C_VEL
LIN {X 0,Y 398.746,Z 1166.208,A -85,B 0,C 180,E1 18670.095,E2 18670.095} C_VEL
LIN {X 0,Y 406.305,Z 1142.254,A -85,B 0,C 180,E1 18673.677,E2 18673.677} C_VEL
LIN {X 0,Y 406.8,Z 1130.679,A -85,B 0,C 180,E1 18675.519,E2 18675.519} C_VEL
LIN {X 0,Y 407.372,Z 1118.698,A -85,B 0,C 180,E1 18677.34,E2 18677.34} C_VEL
LIN {X 0,Y 424.588,Z 1069.327,A -85,B 0,C 180,E1 18682.571,E2 18682.571} C_VEL
LIN {X 0,Y 451.085,Z 1002.143,A -85,B 0,C 180,E1 18687.971,E2 18687.971} C_VEL
LIN {X 0,Y 461,Z 982.117,A -85,B 0,C 180,E1 18689.291,E2 18689.291} C_VEL
LIN {X 0,Y 461.758,Z 980.51,A -85,B 0,C 180,E1 18689.545,E2 18689.545} C_VEL
LIN {X 0,Y 457.95,Z 986.457,A -85,B 0,C 180,E1 18690.606,E2 18690.606} C_VEL
LIN {X 0,Y 433.443,Z 1029.935,A -85,B 0,C 180,E1 18695.584,E2 18695.584} C_VEL
LIN {X 0,Y 413.758,Z 1064.833,A -85,B 0,C 180,E1 18701.088,E2 18701.088} C_VEL
LIN {X 0,Y 397.029,Z 1093.354,A -85,B 0,C 180,E1 18707.288,E2 18707.288} C_VEL
LIN {X 0,Y 384.277,Z 1114.889,A -85,B 0,C 180,E1 18713.792,E2 18713.792} C_VEL
LIN {X 0,Y 375.39,Z 1131.037,A -85,B 0,C 180,E1 18720.576,E2 18720.576} C_VEL
LIN {X 0,Y 369.495,Z 1143.092,A -85,B 0,C 180,E1 18728.228,E2 18728.228} C_VEL
LIN {X 0,Y 366.974,Z 1149.062,A -85,B 0,C 180,E1 18734.302,E2 18734.302} C_VEL
LIN {X 0,Y 365.675,Z 1151.822,A -85,B 0,C 180,E1 18739.302,E2 18739.302} C_VEL
LIN {X 0,Y 365.006,Z 1152.551,A -85,B 0,C 180,E1 18744.453,E2 18744.453} C_VEL
LIN {X 0,Y 365.916,Z 1149.28,A -85,B 0,C 180,E1 18752.466,E2 18752.466} C_VEL
LIN {X 0,Y 367.647,Z 1143.172,A -85,B 0,C 180,E1 18758.672,E2 18758.672} C_VEL
LIN {X 0,Y 371.374,Z 1131.185,A -85,B 0,C 180,E1 18766.249,E2 18766.249} C_VEL
LIN {X 0,Y 378.576,Z 1113.136,A -85,B 0,C 180,E1 18773.697,E2 18773.697} C_VEL
LIN {X 0,Y 388.364,Z 1091.365,A -85,B 0,C 180,E1 18780.16,E2 18780.16} C_VEL
LIN {X 0,Y 401.619,Z 1062.33,A -85,B 0,C 180,E1 18786.422,E2 18786.422} C_VEL
LIN {X 0,Y 415.878,Z 1030.346,A -85,B 0,C 180,E1 18791.544,E2 18791.544} C_VEL
LIN {X 0,Y 432.115,Z 990.566,A -85,B 0,C 180,E1 18796.245,E2 18796.245} C_VEL
LIN {X 0,Y 439.361,Z 971.015,A -85,B 0,C 180,E1 18798.1,E2 18798.1} C_VEL
LIN {X 0,Y 433.336,Z 943.038,A -85,B 0,C 180,E1 18802.998,E2 18802.998} C_VEL
LIN {X 0,Y 424.968,Z 916.359,A -85,B 0,C 180,E1 18807.971,E2 18807.971} C_VEL
LIN {X 0,Y 413.823,Z 889.586,A -85,B 0,C 180,E1 18813.651,E2 18813.651} C_VEL
LIN {X 0,Y 400.719,Z 864.884,A -85,B 0,C 180,E1 18819.976,E2 18819.976} C_VEL
LIN {X 0,Y 387.854,Z 844.368,A -85,B 0,C 180,E1 18826.517,E2 18826.517} C_VEL
LIN {X 0,Y 382.041,Z 836.539,A -85,B 0,C 180,E1 18829.693,E2 18829.693} C_VEL
LIN {X 0,Y 378.04,Z 830.544,A -85,B 0,C 180,E1 18832.162,E2 18832.162} C_VEL
LIN {X 0,Y 374.128,Z 824.442,A -85,B 0,C 180,E1 18834.774,E2 18834.774} C_VEL
LIN {X 0,Y 369.118,Z 818.607,A -85,B 0,C 180,E1 18838.293,E2 18838.293} C_VEL
LIN {X 0,Y 367.887,Z 816.338,A -85,B 0,C 180,E1 18839.294,E2 18839.294} C_VEL
LIN {X 0,Y 363.044,Z 811.169,A -85,B 0,C 180,E1 18843.244,E2 18843.244} C_VEL
LIN {X 0,Y 362.734,Z 809.06,A -85,B 0,C 180,E1 18844.038,E2 18844.038} C_VEL
LIN {X 0,Y 362.688,Z 809.06,A -85,B 0,C 180,E1 18851.42,E2 18851.42} C_VEL
LIN {X 0,Y 362.624,Z 809.06,A -85,B 0,C 180,E1 18858.61,E2 18858.61} C_VEL
LIN {X 0,Y 362.651,Z 809.06,A -85,B 0,C 180,E1 18864.317,E2 18864.317} C_VEL
LIN {X 0,Y 362.997,Z 809.06,A -85,B 0,C 180,E1 18870.966,E2 18870.966} C_VEL
LIN {X 0,Y 363.335,Z 809.06,A -85,B 0,C 180,E1 18878.021,E2 18878.021} C_VEL
LIN {X 0,Y 363.824,Z 809.06,A -85,B 0,C 180,E1 18885.572,E2 18885.572} C_VEL
LIN {X 0,Y 364.019,Z 809.836,A -85,B 0,C 180,E1 18887.575,E2 18887.575} C_VEL
LIN {X 0,Y 366.414,Z 814.64,A -85,B 0,C 180,E1 18889.907,E2 18889.907} C_VEL
LIN {X 0,Y 370.309,Z 817.606,A -85,B 0,C 180,E1 18892.646,E2 18892.646} C_VEL
LIN {X 0,Y 373.862,Z 823.035,A -85,B 0,C 180,E1 18895.181,E2 18895.181} C_VEL
LIN {X 0,Y 376.406,Z 825.512,A -85,B 0,C 180,E1 18896.737,E2 18896.737} C_VEL
LIN {X 0,Y 380.873,Z 831.036,A -85,B 0,C 180,E1 18899.291,E2 18899.291} C_VEL
LIN {X 0,Y 387.947,Z 841.624,A -85,B 0,C 180,E1 18903.071,E2 18903.071} C_VEL
LIN {X 0,Y 396.98,Z 854.064,A -85,B 0,C 180,E1 18907.202,E2 18907.202} C_VEL
LIN {X 0,Y 411.706,Z 875.746,A -85,B 0,C 180,E1 18912.991,E2 18912.991} C_VEL
LIN {X 0,Y 428.475,Z 902.619,A -85,B 0,C 180,E1 18918.806,E2 18918.806} C_VEL
LIN {X 0,Y 445.947,Z 934.631,A -85,B 0,C 180,E1 18924.428,E2 18924.428} C_VEL
LIN {X 0,Y 460.885,Z 967.086,A -85,B 0,C 180,E1 18929.188,E2 18929.188} C_VEL
LIN {X 0,Y 462.97,Z 974.42,A -85,B 0,C 180,E1 18930.067,E2 18930.067} C_VEL
LIN {X 0,Y 449.784,Z 1023.043,A -85,B 0,C 180,E1 18932.458,E2 18932.458} C_VEL
LIN {X 0,Y 434.434,Z 1070.648,A -85,B 0,C 180,E1 18935.807,E2 18935.807} C_VEL
LIN {X 0,Y 419.436,Z 1111.472,A -85,B 0,C 180,E1 18939.689,E2 18939.689} C_VEL
LIN {X 0,Y 404.015,Z 1150.906,A -85,B 0,C 180,E1 18944.703,E2 18944.703} C_VEL
LIN {X 0,Y 390.77,Z 1183.853,A -85,B 0,C 180,E1 18950.278,E2 18950.278} C_VEL
LIN {X 0,Y 379.977,Z 1212.39,A -85,B 0,C 180,E1 18956.625,E2 18956.625} C_VEL
LIN {X 0,Y 372.371,Z 1235.444,A -85,B 0,C 180,E1 18963.478,E2 18963.478} C_VEL
LIN {X 0,Y 367.894,Z 1253.516,A -85,B 0,C 180,E1 18970.849,E2 18970.849} C_VEL
LIN {X 0,Y 366.279,Z 1263.746,A -85,B 0,C 180,E1 18976.876,E2 18976.876} C_VEL
LIN {X 0,Y 365.806,Z 1270.011,A -85,B 0,C 180,E1 18982.872,E2 18982.872} C_VEL
LIN {X 0,Y 365.99,Z 1272.249,A -85,B 0,C 180,E1 18987.624,E2 18987.624} C_VEL
LIN {X 0,Y 366.216,Z 1271.859,A -85,B 0,C 180,E1 18992.355,E2 18992.355} C_VEL
LIN {X 0,Y 366.085,Z 1268.069,A -85,B 0,C 180,E1 18997.863,E2 18997.863} C_VEL
LIN {X 0,Y 366.86,Z 1259.325,A -85,B 0,C 180,E1 19004.298,E2 19004.298} C_VEL
LIN {X 0,Y 368.955,Z 1245.249,A -85,B 0,C 180,E1 19010.926,E2 19010.926} C_VEL
LIN {X 0,Y 373.06,Z 1226.595,A -85,B 0,C 180,E1 19017.282,E2 19017.282} C_VEL
LIN {X 0,Y 380.256,Z 1201.234,A -85,B 0,C 180,E1 19023.791,E2 19023.791} C_VEL
LIN {X 0,Y 390.621,Z 1168.807,A -85,B 0,C 180,E1 19030.107,E2 19030.107} C_VEL
LIN {X 0,Y 403.204,Z 1131.379,A -85,B 0,C 180,E1 19035.737,E2 19035.737} C_VEL
LIN {X 0,Y 407.372,Z 1118.698,A -85,B 0,C 180,E1 19037.34,E2 19037.34} C_VEL
LIN {X 0,Y 408.42,Z 1106.603,A -85,B 0,C 180,E1 19039.125,E2 19039.125} C_VEL
LIN {X 0,Y 410.019,Z 1094.283,A -85,B 0,C 180,E1 19040.851,E2 19040.851} C_VEL
LIN {X 0,Y 432.886,Z 1035.996,A -85,B 0,C 180,E1 19046.351,E2 19046.351} C_VEL
LIN {X 0,Y 452.051,Z 996.638,A -85,B 0,C 180,E1 19049.383,E2 19049.383} C_VEL
LIN {X 0,Y 454.848,Z 991.706,A -85,B 0,C 180,E1 19049.724,E2 19049.724} C_VEL
LIN {X 0,Y 452.787,Z 994.713,A -85,B 0,C 180,E1 19050.237,E2 19050.237} C_VEL
LIN {X 0,Y 426.224,Z 1037.537,A -85,B 0,C 180,E1 19055.462,E2 19055.462} C_VEL
LIN {X 0,Y 406.228,Z 1070.603,A -85,B 0,C 180,E1 19061.006,E2 19061.006} C_VEL
LIN {X 0,Y 389.659,Z 1097.358,A -85,B 0,C 180,E1 19067.116,E2 19067.116} C_VEL
LIN {X 0,Y 375.931,Z 1119.552,A -85,B 0,C 180,E1 19074.232,E2 19074.232} C_VEL
LIN {X 0,Y 366.457,Z 1135.706,A -85,B 0,C 180,E1 19081.771,E2 19081.771} C_VEL
LIN {X 0,Y 361.689,Z 1145.264,A -85,B 0,C 180,E1 19088.407,E2 19088.407} C_VEL
LIN {X 0,Y 359.109,Z 1150.9,A -85,B 0,C 180,E1 19094.622,E2 19094.622} C_VEL
LIN {X 0,Y 357.354,Z 1153.846,A -85,B 0,C 180,E1 19102.366,E2 19102.366} C_VEL
LIN {X 0,Y 357.246,Z 1153.188,A -85,B 0,C 180,E1 19107.725,E2 19107.725} C_VEL
LIN {X 0,Y 358.759,Z 1148.444,A -85,B 0,C 180,E1 19115.154,E2 19115.154} C_VEL
LIN {X 0,Y 361.142,Z 1140.151,A -85,B 0,C 180,E1 19122.022,E2 19122.022} C_VEL
LIN {X 0,Y 366.446,Z 1125.807,A -85,B 0,C 180,E1 19129.717,E2 19129.717} C_VEL
LIN {X 0,Y 375.268,Z 1105.716,A -85,B 0,C 180,E1 19136.982,E2 19136.982} C_VEL
LIN {X 0,Y 386.76,Z 1081.538,A -85,B 0,C 180,E1 19143.372,E2 19143.372} C_VEL
LIN {X 0,Y 401.376,Z 1050.045,A -85,B 0,C 180,E1 19149.416,E2 19149.416} C_VEL
LIN {X 0,Y 416.545,Z 1015.944,A -85,B 0,C 180,E1 19154.257,E2 19154.257} C_VEL
LIN {X 0,Y 432.623,Z 975.517,A -85,B 0,C 180,E1 19158.52,E2 19158.52} C_VEL
LIN {X 0,Y 432.151,Z 968.118,A -85,B 0,C 180,E1 19159.685,E2 19159.685} C_VEL
LIN {X 0,Y 425.733,Z 940.448,A -85,B 0,C 180,E1 19164.739,E2 19164.739} C_VEL
LIN {X 0,Y 417.022,Z 913.797,A -85,B 0,C 180,E1 19170.008,E2 19170.008} C_VEL
LIN {X 0,Y 406.264,Z 889.051,A -85,B 0,C 180,E1 19175.595,E2 19175.595} C_VEL
LIN {X 0,Y 393.751,Z 865.886,A -85,B 0,C 180,E1 19181.995,E2 19181.995} C_VEL
LIN {X 0,Y 384.081,Z 850.598,A -85,B 0,C 180,E1 19187.221,E2 19187.221} C_VEL
LIN {X 0,Y 379.11,Z 843.541,A -85,B 0,C 180,E1 19190.045,E2 19190.045} C_VEL
LIN {X 0,Y 375.219,Z 837.666,A -85,B 0,C 180,E1 19192.539,E2 19192.539} C_VEL
LIN {X 0,Y 370.387,Z 830.767,A -85,B 0,C 180,E1 19195.849,E2 19195.849} C_VEL
LIN {X 0,Y 366.502,Z 825.136,A -85,B 0,C 180,E1 19198.858,E2 19198.858} C_VEL
LIN {X 0,Y 360.916,Z 818.242,A -85,B 0,C 180,E1 19203.688,E2 19203.688} C_VEL
LIN {X 0,Y 360.153,Z 816.493,A -85,B 0,C 180,E1 19204.579,E2 19204.579} C_VEL
LIN {X 0,Y 355.014,Z 811.291,A -85,B 0,C 180,E1 19210.484,E2 19210.484} C_VEL
LIN {X 0,Y 354.785,Z 809.06,A -85,B 0,C 180,E1 19211.623,E2 19211.623} C_VEL
LIN {X 0,Y 354.591,Z 809.06,A -85,B 0,C 180,E1 19217.017,E2 19217.017} C_VEL
LIN {X 0,Y 354.749,Z 809.06,A -85,B 0,C 180,E1 19224.045,E2 19224.045} C_VEL
LIN {X 0,Y 355.105,Z 809.06,A -85,B 0,C 180,E1 19232.093,E2 19232.093} C_VEL
LIN {X 0,Y 355.512,Z 809.503,A -85,B 0,C 180,E1 19239.865,E2 19239.865} C_VEL
LIN {X 0,Y 357.861,Z 814.411,A -85,B 0,C 180,E1 19243.285,E2 19243.285} C_VEL
LIN {X 0,Y 362.123,Z 817.69,A -85,B 0,C 180,E1 19247.333,E2 19247.333} C_VEL
LIN {X 0,Y 365.436,Z 822.892,A -85,B 0,C 180,E1 19250.331,E2 19250.331} C_VEL
LIN {X 0,Y 368.453,Z 825.469,A -85,B 0,C 180,E1 19252.445,E2 19252.445} C_VEL
LIN {X 0,Y 372.622,Z 831.022,A -85,B 0,C 180,E1 19255.349,E2 19255.349} C_VEL
LIN {X 0,Y 374.687,Z 833.765,A -85,B 0,C 180,E1 19256.678,E2 19256.678} C_VEL
LIN {X 0,Y 380.199,Z 841.001,A -85,B 0,C 180,E1 19259.859,E2 19259.859} C_VEL
LIN {X 0,Y 386.171,Z 849.697,A -85,B 0,C 180,E1 19263.015,E2 19263.015} C_VEL
LIN {X 0,Y 396.265,Z 863.941,A -85,B 0,C 180,E1 19267.663,E2 19267.663} C_VEL
LIN {X 0,Y 410.569,Z 885.399,A -85,B 0,C 180,E1 19273.366,E2 19273.366} C_VEL
LIN {X 0,Y 427.295,Z 913.509,A -85,B 0,C 180,E1 19279.295,E2 19279.295} C_VEL
LIN {X 0,Y 444.085,Z 945.897,A -85,B 0,C 180,E1 19284.902,E2 19284.902} C_VEL
LIN {X 0,Y 457.158,Z 975.917,A -85,B 0,C 180,E1 19289.322,E2 19289.322} C_VEL
LIN {X 0,Y 444.249,Z 1023.258,A -85,B 0,C 180,E1 19291.737,E2 19291.737} C_VEL
LIN {X 0,Y 428.241,Z 1071.522,A -85,B 0,C 180,E1 19295.172,E2 19295.172} C_VEL
LIN {X 0,Y 412.686,Z 1112.525,A -85,B 0,C 180,E1 19299.141,E2 19299.141} C_VEL
LIN {X 0,Y 397.276,Z 1150.709,A -85,B 0,C 180,E1 19304.085,E2 19304.085} C_VEL
LIN {X 0,Y 383.07,Z 1184.961,A -85,B 0,C 180,E1 19310.029,E2 19310.029} C_VEL
LIN {X 0,Y 372.103,Z 1213.101,A -85,B 0,C 180,E1 19316.503,E2 19316.503} C_VEL
LIN {X 0,Y 364.377,Z 1235.738,A -85,B 0,C 180,E1 19323.515,E2 19323.515} C_VEL
LIN {X 0,Y 359.936,Z 1253.471,A -85,B 0,C 180,E1 19331.058,E2 19331.058} C_VEL
LIN {X 0,Y 358.302,Z 1264.066,A -85,B 0,C 180,E1 19337.817,E2 19337.817} C_VEL
LIN {X 0,Y 357.981,Z 1268.73,A -85,B 0,C 180,E1 19342.715,E2 19342.715} C_VEL
LIN {X 0,Y 358.176,Z 1270.961,A -85,B 0,C 180,E1 19347.572,E2 19347.572} C_VEL
LIN {X 0,Y 358.419,Z 1270.54,A -85,B 0,C 180,E1 19352.406,E2 19352.406} C_VEL
LIN {X 0,Y 358.264,Z 1266.694,A -85,B 0,C 180,E1 19358.036,E2 19358.036} C_VEL
LIN {X 0,Y 359.101,Z 1257.843,A -85,B 0,C 180,E1 19364.614,E2 19364.614} C_VEL
LIN {X 0,Y 361.306,Z 1243.52,A -85,B 0,C 180,E1 19371.455,E2 19371.455} C_VEL
LIN {X 0,Y 366.036,Z 1223.404,A -85,B 0,C 180,E1 19378.331,E2 19378.331} C_VEL
LIN {X 0,Y 373.936,Z 1196.989,A -85,B 0,C 180,E1 19385.035,E2 19385.035} C_VEL
LIN {X 0,Y 385.099,Z 1163.844,A -85,B 0,C 180,E1 19391.451,E2 19391.451} C_VEL
LIN {X 0,Y 398.697,Z 1125.115,A -85,B 0,C 180,E1 19397.204,E2 19397.204} C_VEL
LIN {X 0,Y 410.019,Z 1094.283,A -85,B 0,C 180,E1 19400.851,E2 19400.851} C_VEL
LIN {X 0,Y 411.99,Z 1081.976,A -85,B 0,C 180,E1 19402.569,E2 19402.569} C_VEL
LIN {X 0,Y 414.252,Z 1069.607,A -85,B 0,C 180,E1 19404.264,E2 19404.264} C_VEL
LIN {X 0,Y 441.359,Z 1013.169,A -85,B 0,C 180,E1 19409.265,E2 19409.265} C_VEL
LIN {X 0,Y 445.954,Z 1005.467,A -85,B 0,C 180,E1 19409.843,E2 19409.843} C_VEL
LIN {X 0,Y 446.45,Z 1004.489,A -85,B 0,C 180,E1 19410.051,E2 19410.051} C_VEL
LIN {X 0,Y 419.462,Z 1044.453,A -85,B 0,C 180,E1 19415.243,E2 19415.243} C_VEL
LIN {X 0,Y 397.215,Z 1078.842,A -85,B 0,C 180,E1 19421.422,E2 19421.422} C_VEL
LIN {X 0,Y 378.812,Z 1106.679,A -85,B 0,C 180,E1 19428.495,E2 19428.495} C_VEL
LIN {X 0,Y 364.981,Z 1128.04,A -85,B 0,C 180,E1 19436.439,E2 19436.439} C_VEL
LIN {X 0,Y 357.302,Z 1140.868,A -85,B 0,C 180,E1 19443.488,E2 19443.488} C_VEL
LIN {X 0,Y 353.088,Z 1148.999,A -85,B 0,C 180,E1 19450.227,E2 19450.227} C_VEL
LIN {X 0,Y 350.465,Z 1154.011,A -85,B 0,C 180,E1 19457.565,E2 19457.565} C_VEL
LIN {X 0,Y 349.356,Z 1154.978,A -85,B 0,C 180,E1 19465.626,E2 19465.626} C_VEL
LIN {X 0,Y 350.47,Z 1151.46,A -85,B 0,C 180,E1 19473.118,E2 19473.118} C_VEL
LIN {X 0,Y 352.55,Z 1144.534,A -85,B 0,C 180,E1 19480.006,E2 19480.006} C_VEL
LIN {X 0,Y 356.55,Z 1132.89,A -85,B 0,C 180,E1 19487.32,E2 19487.32} C_VEL
LIN {X 0,Y 364.679,Z 1114.422,A -85,B 0,C 180,E1 19495.027,E2 19495.027} C_VEL
LIN {X 0,Y 375.224,Z 1092.399,A -85,B 0,C 180,E1 19501.642,E2 19501.642} C_VEL
LIN {X 0,Y 389.699,Z 1062.593,A -85,B 0,C 180,E1 19508.104,E2 19508.104} C_VEL
LIN {X 0,Y 404.779,Z 1030.411,A -85,B 0,C 180,E1 19513.241,E2 19513.241} C_VEL
LIN {X 0,Y 421.31,Z 991.637,A -85,B 0,C 180,E1 19517.824,E2 19517.824} C_VEL
LIN {X 0,Y 426.89,Z 976.652,A -85,B 0,C 180,E1 19519.298,E2 19519.298} C_VEL
LIN {X 0,Y 421.222,Z 949.108,A -85,B 0,C 180,E1 19524.399,E2 19524.399} C_VEL
LIN {X 0,Y 413.128,Z 922.319,A -85,B 0,C 180,E1 19529.747,E2 19529.747} C_VEL
LIN {X 0,Y 403.153,Z 897.502,A -85,B 0,C 180,E1 19535.385,E2 19535.385} C_VEL
LIN {X 0,Y 391.468,Z 875.04,A -85,B 0,C 180,E1 19541.557,E2 19541.557} C_VEL
LIN {X 0,Y 381.891,Z 858.689,A -85,B 0,C 180,E1 19546.985,E2 19546.985} C_VEL
LIN {X 0,Y 372.372,Z 844.827,A -85,B 0,C 180,E1 19552.87,E2 19552.87} C_VEL
LIN {X 0,Y 367.623,Z 837.886,A -85,B 0,C 180,E1 19556.327,E2 19556.327} C_VEL
LIN {X 0,Y 363.9,Z 831.759,A -85,B 0,C 180,E1 19559.396,E2 19559.396} C_VEL
LIN {X 0,Y 358.845,Z 825.75,A -85,B 0,C 180,E1 19563.951,E2 19563.951} C_VEL
LIN {X 0,Y 357.699,Z 823.906,A -85,B 0,C 180,E1 19565.301,E2 19565.301} C_VEL
LIN {X 0,Y 353.06,Z 818.393,A -85,B 0,C 180,E1 19570.961,E2 19570.961} C_VEL
LIN {X 0,Y 352.663,Z 816.678,A -85,B 0,C 180,E1 19571.945,E2 19571.945} C_VEL
LIN {X 0,Y 348.419,Z 813.83,A -85,B 0,C 180,E1 19583.286,E2 19583.286} C_VEL
LIN {X 0,Y 349.75,Z 814.846,A -85,B 0,C 180,E1 19592.667,E2 19592.667} C_VEL
LIN {X 0,Y 353.861,Z 817.701,A -85,B 0,C 180,E1 19599.852,E2 19599.852} C_VEL
LIN {X 0,Y 357.008,Z 822.883,A -85,B 0,C 180,E1 19604.033,E2 19604.033} C_VEL
LIN {X 0,Y 360.258,Z 825.443,A -85,B 0,C 180,E1 19607.092,E2 19607.092} C_VEL
LIN {X 0,Y 364.205,Z 830.89,A -85,B 0,C 180,E1 19610.552,E2 19610.552} C_VEL
LIN {X 0,Y 366.573,Z 833.244,A -85,B 0,C 180,E1 19612.243,E2 19612.243} C_VEL
LIN {X 0,Y 371.316,Z 838.962,A -85,B 0,C 180,E1 19615.479,E2 19615.479} C_VEL
LIN {X 0,Y 378.136,Z 848.638,A -85,B 0,C 180,E1 19619.65,E2 19619.65} C_VEL
LIN {X 0,Y 387.826,Z 862.581,A -85,B 0,C 180,E1 19624.68,E2 19624.68} C_VEL
LIN {X 0,Y 400.348,Z 881.283,A -85,B 0,C 180,E1 19630.226,E2 19630.226} C_VEL
LIN {X 0,Y 414.928,Z 904.842,A -85,B 0,C 180,E1 19635.879,E2 19635.879} C_VEL
LIN {X 0,Y 431.171,Z 934.522,A -85,B 0,C 180,E1 19641.658,E2 19641.658} C_VEL
LIN {X 0,Y 446.985,Z 968.518,A -85,B 0,C 180,E1 19647.156,E2 19647.156} C_VEL
LIN {X 0,Y 451.142,Z 980.831,A -85,B 0,C 180,E1 19648.807,E2 19648.807} C_VEL
LIN {X 0,Y 437.132,Z 1028.403,A -85,B 0,C 180,E1 19651.297,E2 19651.297} C_VEL
LIN {X 0,Y 421.538,Z 1073.895,A -85,B 0,C 180,E1 19654.647,E2 19654.647} C_VEL
LIN {X 0,Y 404.411,Z 1117.461,A -85,B 0,C 180,E1 19659.04,E2 19659.04} C_VEL
LIN {X 0,Y 389.057,Z 1154.058,A -85,B 0,C 180,E1 19664.015,E2 19664.015} C_VEL
LIN {X 0,Y 374.494,Z 1188.278,A -85,B 0,C 180,E1 19670.234,E2 19670.234} C_VEL
LIN {X 0,Y 363.481,Z 1215.54,A -85,B 0,C 180,E1 19676.91,E2 19676.91} C_VEL
LIN {X 0,Y 355.839,Z 1238.001,A -85,B 0,C 180,E1 19684.297,E2 19684.297} C_VEL
LIN {X 0,Y 351.866,Z 1253.841,A -85,B 0,C 180,E1 19691.595,E2 19691.595} C_VEL
LIN {X 0,Y 350.362,Z 1264.114,A -85,B 0,C 180,E1 19698.799,E2 19698.799} C_VEL
LIN {X 0,Y 350.187,Z 1268.844,A -85,B 0,C 180,E1 19705.039,E2 19705.039} C_VEL
LIN {X 0,Y 350.649,Z 1269.862,A -85,B 0,C 180,E1 19709.99,E2 19709.99} C_VEL
LIN {X 0,Y 350.445,Z 1267.962,A -85,B 0,C 180,E1 19714.937,E2 19714.937} C_VEL
LIN {X 0,Y 350.642,Z 1261.974,A -85,B 0,C 180,E1 19721.171,E2 19721.171} C_VEL
LIN {X 0,Y 351.855,Z 1251.756,A -85,B 0,C 180,E1 19727.484,E2 19727.484} C_VEL
LIN {X 0,Y 355.187,Z 1235.065,A -85,B 0,C 180,E1 19734.558,E2 19734.558} C_VEL
LIN {X 0,Y 361.952,Z 1210.933,A -85,B 0,C 180,E1 19741.976,E2 19741.976} C_VEL
LIN {X 0,Y 371.781,Z 1181.135,A -85,B 0,C 180,E1 19748.769,E2 19748.769} C_VEL
LIN {X 0,Y 385.307,Z 1143.79,A -85,B 0,C 180,E1 19755.246,E2 19755.246} C_VEL
LIN {X 0,Y 401.731,Z 1100.528,A -85,B 0,C 180,E1 19760.942,E2 19760.942} C_VEL
LIN {X 0,Y 414.252,Z 1069.607,A -85,B 0,C 180,E1 19764.264,E2 19764.264} C_VEL
LIN {X 0,Y 417.489,Z 1057.415,A -85,B 0,C 180,E1 19765.953,E2 19765.953} C_VEL
LIN {X 0,Y 420.732,Z 1046.855,A -85,B 0,C 180,E1 19767.406,E2 19767.406} C_VEL
LIN {X 0,Y 421.572,Z 1045.214,A -85,B 0,C 180,E1 19767.565,E2 19767.565} C_VEL
LIN {X 0,Y 436.585,Z 1019.131,A -85,B 0,C 180,E1 19769.897,E2 19769.897} C_VEL
LIN {X 0,Y 437.614,Z 1017.303,A -85,B 0,C 180,E1 19770.238,E2 19770.238} C_VEL
LIN {X 0,Y 409.584,Z 1055.721,A -85,B 0,C 180,E1 19775.768,E2 19775.768} C_VEL
LIN {X 0,Y 388.105,Z 1086.562,A -85,B 0,C 180,E1 19781.852,E2 19781.852} C_VEL
LIN {X 0,Y 370.487,Z 1111.632,A -85,B 0,C 180,E1 19788.748,E2 19788.748} C_VEL
LIN {X 0,Y 357.44,Z 1130.833,A -85,B 0,C 180,E1 19796.32,E2 19796.32} C_VEL
LIN {X 0,Y 348.465,Z 1145.218,A -85,B 0,C 180,E1 19804.974,E2 19804.974} C_VEL
LIN {X 0,Y 344.266,Z 1152.799,A -85,B 0,C 180,E1 19812.676,E2 19812.676} C_VEL
LIN {X 0,Y 342.007,Z 1156.336,A -85,B 0,C 180,E1 19820.697,E2 19820.697} C_VEL
LIN {X 0,Y 341.782,Z 1155.173,A -85,B 0,C 180,E1 19829.097,E2 19829.097} C_VEL
LIN {X 0,Y 343.369,Z 1150.369,A -85,B 0,C 180,E1 19836.021,E2 19836.021} C_VEL
LIN {X 0,Y 346.062,Z 1141.898,A -85,B 0,C 180,E1 19843.035,E2 19843.035} C_VEL
LIN {X 0,Y 351.726,Z 1127.992,A -85,B 0,C 180,E1 19850.647,E2 19850.647} C_VEL
LIN {X 0,Y 361.231,Z 1107.865,A -85,B 0,C 180,E1 19858.126,E2 19858.126} C_VEL
LIN {X 0,Y 373.717,Z 1083.153,A -85,B 0,C 180,E1 19864.776,E2 19864.776} C_VEL
LIN {X 0,Y 389.035,Z 1052.082,A -85,B 0,C 180,E1 19870.842,E2 19870.842} C_VEL
LIN {X 0,Y 404.672,Z 1018.653,A -85,B 0,C 180,E1 19875.656,E2 19875.656} C_VEL
LIN {X 0,Y 420.615,Z 979.517,A -85,B 0,C 180,E1 19879.922,E2 19879.922} C_VEL
LIN {X 0,Y 414.982,Z 951.283,A -85,B 0,C 180,E1 19885.309,E2 19885.309} C_VEL
LIN {X 0,Y 407.417,Z 925.705,A -85,B 0,C 180,E1 19890.568,E2 19890.568} C_VEL
LIN {X 0,Y 397.86,Z 901.565,A -85,B 0,C 180,E1 19896.257,E2 19896.257} C_VEL
LIN {X 0,Y 386.804,Z 879.912,A -85,B 0,C 180,E1 19902.427,E2 19902.427} C_VEL
LIN {X 0,Y 376.883,Z 863.393,A -85,B 0,C 180,E1 19908.292,E2 19908.292} C_VEL
LIN {X 0,Y 369.034,Z 851.345,A -85,B 0,C 180,E1 19913.538,E2 19913.538} C_VEL
LIN {X 0,Y 364.814,Z 844.987,A -85,B 0,C 180,E1 19916.712,E2 19916.712} C_VEL
LIN {X 0,Y 360.426,Z 838.434,A -85,B 0,C 180,E1 19920.511,E2 19920.511} C_VEL
LIN {X 0,Y 356.426,Z 832.395,A -85,B 0,C 180,E1 19924.534,E2 19924.534} C_VEL
LIN {X 0,Y 351.212,Z 825.955,A -85,B 0,C 180,E1 19931.201,E2 19931.201} C_VEL
LIN {X 0,Y 350.387,Z 824.212,A -85,B 0,C 180,E1 19932.855,E2 19932.855} C_VEL
LIN {X 0,Y 346.778,Z 821.482,A -85,B 0,C 180,E1 19943.887,E2 19943.887} C_VEL
LIN {X 0,Y 348.267,Z 822.68,A -85,B 0,C 180,E1 19952.87,E2 19952.87} C_VEL
LIN {X 0,Y 352.174,Z 825.416,A -85,B 0,C 180,E1 19959.681,E2 19959.681} C_VEL
LIN {X 0,Y 355.556,Z 830.688,A -85,B 0,C 180,E1 19964.124,E2 19964.124} C_VEL
LIN {X 0,Y 358.468,Z 833.083,A -85,B 0,C 180,E1 19966.884,E2 19966.884} C_VEL
LIN {X 0,Y 362.419,Z 838.5,A -85,B 0,C 180,E1 19970.401,E2 19970.401} C_VEL
LIN {X 0,Y 364.702,Z 841.177,A -85,B 0,C 180,E1 19972.121,E2 19972.121} C_VEL
LIN {X 0,Y 370.564,Z 848.706,A -85,B 0,C 180,E1 19976.147,E2 19976.147} C_VEL
LIN {X 0,Y 376.386,Z 856.801,A -85,B 0,C 180,E1 19979.656,E2 19979.656} C_VEL
LIN {X 0,Y 385.922,Z 870.773,A -85,B 0,C 180,E1 19984.703,E2 19984.703} C_VEL
LIN {X 0,Y 398.827,Z 890.549,A -85,B 0,C 180,E1 19990.494,E2 19990.494} C_VEL
LIN {X 0,Y 413.205,Z 914.56,A -85,B 0,C 180,E1 19996.2,E2 19996.2} C_VEL
LIN {X 0,Y 428.757,Z 944.546,A -85,B 0,C 180,E1 20001.99,E2 20001.99} C_VEL
LIN {X 0,Y 442.409,Z 975.075,A -85,B 0,C 180,E1 20006.962,E2 20006.962} C_VEL
LIN {X 0,Y 445.472,Z 982.886,A -85,B 0,C 180,E1 20008.108,E2 20008.108} C_VEL
LIN {X 0,Y 430.273,Z 1032.926,A -85,B 0,C 180,E1 20010.831,E2 20010.831} C_VEL
LIN {X 0,Y 414.635,Z 1076.561,A -85,B 0,C 180,E1 20014.146,E2 20014.146} C_VEL
LIN {X 0,Y 397.199,Z 1119.563,A -85,B 0,C 180,E1 20018.595,E2 20018.595} C_VEL
LIN {X 0,Y 380.755,Z 1157.414,A -85,B 0,C 180,E1 20023.96,E2 20023.96} C_VEL
LIN {X 0,Y 366.733,Z 1189.353,A -85,B 0,C 180,E1 20030.001,E2 20030.001} C_VEL
LIN {X 0,Y 354.77,Z 1218.299,A -85,B 0,C 180,E1 20037.438,E2 20037.438} C_VEL
LIN {X 0,Y 347.485,Z 1239.229,A -85,B 0,C 180,E1 20044.806,E2 20044.806} C_VEL
LIN {X 0,Y 343.666,Z 1255.079,A -85,B 0,C 180,E1 20052.725,E2 20052.725} C_VEL
LIN {X 0,Y 342.49,Z 1264.15,A -85,B 0,C 180,E1 20059.825,E2 20059.825} C_VEL
LIN {X 0,Y 342.563,Z 1268.398,A -85,B 0,C 180,E1 20067.462,E2 20067.462} C_VEL
LIN {X 0,Y 342.808,Z 1267.907,A -85,B 0,C 180,E1 20072.516,E2 20072.516} C_VEL
LIN {X 0,Y 342.65,Z 1263.483,A -85,B 0,C 180,E1 20078.868,E2 20078.868} C_VEL
LIN {X 0,Y 343.496,Z 1254.926,A -85,B 0,C 180,E1 20085.293,E2 20085.293} C_VEL
LIN {X 0,Y 346.011,Z 1240.33,A -85,B 0,C 180,E1 20092.454,E2 20092.454} C_VEL
LIN {X 0,Y 351.333,Z 1219.951,A -85,B 0,C 180,E1 20099.632,E2 20099.632} C_VEL
LIN {X 0,Y 359.77,Z 1194.246,A -85,B 0,C 180,E1 20106.397,E2 20106.397} C_VEL
LIN {X 0,Y 372.213,Z 1160.434,A -85,B 0,C 180,E1 20113.159,E2 20113.159} C_VEL
LIN {X 0,Y 388.159,Z 1119.716,A -85,B 0,C 180,E1 20119.371,E2 20119.371} C_VEL
LIN {X 0,Y 415.434,Z 1057.212,A -85,B 0,C 180,E1 20126.425,E2 20126.425} C_VEL
LIN {X 0,Y 421.572,Z 1045.214,A -85,B 0,C 180,E1 20127.565,E2 20127.565} C_VEL
LIN {X 0,Y 424.435,Z 1038.04,A -85,B 0,C 180,E1 20128.781,E2 20128.781} C_VEL
LIN {X 0,Y 427.717,Z 1031.073,A -85,B 0,C 180,E1 20129.993,E2 20129.993} C_VEL
LIN {X 0,Y 428.615,Z 1029.39,A -85,B 0,C 180,E1 20130.426,E2 20130.426} C_VEL
LIN {X 0,Y 397.63,Z 1068.993,A -85,B 0,C 180,E1 20136.78,E2 20136.78} C_VEL
LIN {X 0,Y 376.726,Z 1097.117,A -85,B 0,C 180,E1 20143.094,E2 20143.094} C_VEL
LIN {X 0,Y 359.592,Z 1120.129,A -85,B 0,C 180,E1 20150.323,E2 20150.323} C_VEL
LIN {X 0,Y 346.808,Z 1138.121,A -85,B 0,C 180,E1 20158.626,E2 20158.626} C_VEL
LIN {X 0,Y 338.971,Z 1150.364,A -85,B 0,C 180,E1 20167.684,E2 20167.684} C_VEL
LIN {X 0,Y 335.44,Z 1156.182,A -85,B 0,C 180,E1 20175.679,E2 20175.679} C_VEL
LIN {X 0,Y 334.126,Z 1157.849,A -85,B 0,C 180,E1 20181.208,E2 20181.208} C_VEL
LIN {X 0,Y 333.752,Z 1157.256,A -85,B 0,C 180,E1 20186.918,E2 20186.918} C_VEL
LIN {X 0,Y 335.053,Z 1153.516,A -85,B 0,C 180,E1 20193.963,E2 20193.963} C_VEL
LIN {X 0,Y 337.472,Z 1146.164,A -85,B 0,C 180,E1 20201.175,E2 20201.175} C_VEL
LIN {X 0,Y 342.519,Z 1132.94,A -85,B 0,C 180,E1 20209.242,E2 20209.242} C_VEL
LIN {X 0,Y 351.725,Z 1114.129,A -85,B 0,C 180,E1 20217.027,E2 20217.027} C_VEL
LIN {X 0,Y 364.085,Z 1089.932,A -85,B 0,C 180,E1 20224.067,E2 20224.067} C_VEL
LIN {X 0,Y 378.99,Z 1061.124,A -85,B 0,C 180,E1 20230.182,E2 20230.182} C_VEL
LIN {X 0,Y 395.481,Z 1027.112,A -85,B 0,C 180,E1 20235.451,E2 20235.451} C_VEL
LIN {X 0,Y 411.558,Z 990.741,A -85,B 0,C 180,E1 20239.672,E2 20239.672} C_VEL
LIN {X 0,Y 414.435,Z 982.921,A -85,B 0,C 180,E1 20240.459,E2 20240.459} C_VEL
LIN {X 0,Y 409.301,Z 955.743,A -85,B 0,C 180,E1 20245.774,E2 20245.774} C_VEL
LIN {X 0,Y 402.272,Z 930.623,A -85,B 0,C 180,E1 20251.085,E2 20251.085} C_VEL
LIN {X 0,Y 393.394,Z 907.549,A -85,B 0,C 180,E1 20256.626,E2 20256.626} C_VEL
LIN {X 0,Y 382.534,Z 885.286,A -85,B 0,C 180,E1 20263.143,E2 20263.143} C_VEL
LIN {X 0,Y 371.928,Z 866.977,A -85,B 0,C 180,E1 20269.824,E2 20269.824} C_VEL
LIN {X 0,Y 362.424,Z 852.512,A -85,B 0,C 180,E1 20276.79,E2 20276.79} C_VEL
LIN {X 0,Y 357.794,Z 845.699,A -85,B 0,C 180,E1 20280.897,E2 20280.897} C_VEL
LIN {X 0,Y 353.387,Z 839.002,A -85,B 0,C 180,E1 20285.672,E2 20285.672} C_VEL
LIN {X 0,Y 349.17,Z 833.295,A -85,B 0,C 180,E1 20291.536,E2 20291.536} C_VEL
LIN {X 0,Y 348.804,Z 831.956,A -85,B 0,C 180,E1 20292.574,E2 20292.574} C_VEL
LIN {X 0,Y 345.097,Z 829.207,A -85,B 0,C 180,E1 20303.683,E2 20303.683} C_VEL
LIN {X 0,Y 346.529,Z 830.345,A -85,B 0,C 180,E1 20312.722,E2 20312.722} C_VEL
LIN {X 0,Y 350.369,Z 832.999,A -85,B 0,C 180,E1 20319.445,E2 20319.445} C_VEL
LIN {X 0,Y 353.77,Z 838.325,A -85,B 0,C 180,E1 20324.021,E2 20324.021} C_VEL
LIN {X 0,Y 356.532,Z 840.798,A -85,B 0,C 180,E1 20326.691,E2 20326.691} C_VEL
LIN {X 0,Y 361.09,Z 846.463,A -85,B 0,C 180,E1 20330.669,E2 20330.669} C_VEL
LIN {X 0,Y 368.521,Z 856.401,A -85,B 0,C 180,E1 20335.968,E2 20335.968} C_VEL
LIN {X 0,Y 374.391,Z 864.646,A -85,B 0,C 180,E1 20339.567,E2 20339.567} C_VEL
LIN {X 0,Y 385.859,Z 881.684,A -85,B 0,C 180,E1 20345.673,E2 20345.673} C_VEL
LIN {X 0,Y 399.447,Z 903.711,A -85,B 0,C 180,E1 20351.831,E2 20351.831} C_VEL
LIN {X 0,Y 414.273,Z 930.232,A -85,B 0,C 180,E1 20357.787,E2 20357.787} C_VEL
LIN {X 0,Y 429.57,Z 961.748,A -85,B 0,C 180,E1 20363.587,E2 20363.587} C_VEL
LIN {X 0,Y 439.355,Z 986.727,A -85,B 0,C 180,E1 20367.503,E2 20367.503} C_VEL
LIN {X 0,Y 424.051,Z 1035.348,A -85,B 0,C 180,E1 20370.206,E2 20370.206} C_VEL
LIN {X 0,Y 406.883,Z 1081.171,A -85,B 0,C 180,E1 20373.814,E2 20373.814} C_VEL
LIN {X 0,Y 390.336,Z 1120.746,A -85,B 0,C 180,E1 20378.042,E2 20378.042} C_VEL
LIN {X 0,Y 372.94,Z 1159.499,A -85,B 0,C 180,E1 20383.695,E2 20383.695} C_VEL
LIN {X 0,Y 358.873,Z 1190.513,A -85,B 0,C 180,E1 20389.799,E2 20389.799} C_VEL
LIN {X 0,Y 346.817,Z 1218.923,A -85,B 0,C 180,E1 20397.361,E2 20397.361} C_VEL
LIN {X 0,Y 339.428,Z 1239.516,A -85,B 0,C 180,E1 20404.97,E2 20404.97} C_VEL
LIN {X 0,Y 335.753,Z 1254.792,A -85,B 0,C 180,E1 20412.979,E2 20412.979} C_VEL
LIN {X 0,Y 334.682,Z 1262.823,A -85,B 0,C 180,E1 20419.585,E2 20419.585} C_VEL
LIN {X 0,Y 334.579,Z 1266.263,A -85,B 0,C 180,E1 20424.807,E2 20424.807} C_VEL
LIN {X 0,Y 335.08,Z 1267.249,A -85,B 0,C 180,E1 20429.989,E2 20429.989} C_VEL
LIN {X 0,Y 334.752,Z 1264.235,A -85,B 0,C 180,E1 20436.762,E2 20436.762} C_VEL
LIN {X 0,Y 335.417,Z 1256.407,A -85,B 0,C 180,E1 20443.816,E2 20443.816} C_VEL
LIN {X 0,Y 337.419,Z 1243.373,A -85,B 0,C 180,E1 20450.982,E2 20450.982} C_VEL
LIN {X 0,Y 342.425,Z 1223.353,A -85,B 0,C 180,E1 20458.672,E2 20458.672} C_VEL
LIN {X 0,Y 351.117,Z 1197.461,A -85,B 0,C 180,E1 20466.024,E2 20466.024} C_VEL
LIN {X 0,Y 363.394,Z 1165.434,A -85,B 0,C 180,E1 20472.874,E2 20472.874} C_VEL
LIN {X 0,Y 380.664,Z 1123.132,A -85,B 0,C 180,E1 20479.699,E2 20479.699} C_VEL
LIN {X 0,Y 410.725,Z 1059.567,A -85,B 0,C 180,E1 20487.241,E2 20487.241} C_VEL
LIN {X 0,Y 427.717,Z 1031.073,A -85,B 0,C 180,E1 20489.993,E2 20489.993} C_VEL
LIN {X 0,Y 426.188,Z 1032.612,A -85,B 0,C 180,E1 20490.47,E2 20490.47} C_VEL
LIN {X 0,Y 414.218,Z 1046.912,A -85,B 0,C 180,E1 20491.536,E2 20491.536} C_VEL
LIN {X 0,Y 384.702,Z 1082.596,A -85,B 0,C 180,E1 20498.15,E2 20498.15} C_VEL
LIN {X 0,Y 363.864,Z 1108.738,A -85,B 0,C 180,E1 20504.956,E2 20504.956} C_VEL
LIN {X 0,Y 347.905,Z 1129.084,A -85,B 0,C 180,E1 20512.513,E2 20512.513} C_VEL
LIN {X 0,Y 337.482,Z 1142.965,A -85,B 0,C 180,E1 20519.999,E2 20519.999} C_VEL
LIN {X 0,Y 331.147,Z 1152.504,A -85,B 0,C 180,E1 20527.867,E2 20527.867} C_VEL
LIN {X 0,Y 327.526,Z 1157.869,A -85,B 0,C 180,E1 20536.068,E2 20536.068} C_VEL
LIN {X 0,Y 325.958,Z 1159.138,A -85,B 0,C 180,E1 20544.657,E2 20544.657} C_VEL
LIN {X 0,Y 326.397,Z 1157.032,A -85,B 0,C 180,E1 20550.611,E2 20550.611} C_VEL
LIN {X 0,Y 328.028,Z 1152.442,A -85,B 0,C 180,E1 20556.784,E2 20556.784} C_VEL
LIN {X 0,Y 331.264,Z 1143.196,A -85,B 0,C 180,E1 20564.439,E2 20564.439} C_VEL
LIN {X 0,Y 337.613,Z 1129.009,A -85,B 0,C 180,E1 20572.126,E2 20572.126} C_VEL
LIN {X 0,Y 348.614,Z 1107.669,A -85,B 0,C 180,E1 20580.093,E2 20580.093} C_VEL
LIN {X 0,Y 361.915,Z 1082.744,A -85,B 0,C 180,E1 20586.705,E2 20586.705} C_VEL
LIN {X 0,Y 378.733,Z 1050.493,A -85,B 0,C 180,E1 20592.954,E2 20592.954} C_VEL
LIN {X 0,Y 396.191,Z 1014.223,A -85,B 0,C 180,E1 20597.997,E2 20597.997} C_VEL
LIN {X 0,Y 407.932,Z 987.266,A -85,B 0,C 180,E1 20600.898,E2 20600.898} C_VEL
LIN {X 0,Y 404.779,Z 965.382,A -85,B 0,C 180,E1 20605.191,E2 20605.191} C_VEL
LIN {X 0,Y 398.603,Z 940.691,A -85,B 0,C 180,E1 20610.414,E2 20610.414} C_VEL
LIN {X 0,Y 390.164,Z 916.355,A -85,B 0,C 180,E1 20616.261,E2 20616.261} C_VEL
LIN {X 0,Y 379.925,Z 894.355,A -85,B 0,C 180,E1 20622.645,E2 20622.645} C_VEL
LIN {X 0,Y 371.098,Z 878.321,A -85,B 0,C 180,E1 20628.38,E2 20628.38} C_VEL
LIN {X 0,Y 363.518,Z 865.974,A -85,B 0,C 180,E1 20633.875,E2 20633.875} C_VEL
LIN {X 0,Y 355.821,Z 853.504,A -85,B 0,C 180,E1 20640.648,E2 20640.648} C_VEL
LIN {X 0,Y 351.802,Z 847.027,A -85,B 0,C 180,E1 20645.178,E2 20645.178} C_VEL
